METHOD _copyFromModel_SM_ConfigManager
  VAR_IN_OUT
    {attribute 'OPC.UA.DA' := '0'}
    model : M_SM_ConfigManager;
  END_VAR
                  THIS^.proc.save._copyFromModel_WriteXmlProcess( model := model.proc.save );
THIS^.proc.load._copyFromModel_ReadXmlProcess( model := model.proc.load );
THIS^.proc.activate._copyFromModel_ActivateProcess( model := model.proc.activate );

                
END_METHOD

METHOD _copyToModel_SM_ConfigManager
  VAR_IN_OUT
    {attribute 'OPC.UA.DA' := '0'}
    model : M_SM_ConfigManager;
  END_VAR
                  model.filePath := THIS^.filePath;
model.actualStatus := THIS^.actualStatus;
model.stat := THIS^.stat;
THIS^.proc.save._copyToModel_WriteXmlProcess( model := model.proc.save );
THIS^.proc.load._copyToModel_ReadXmlProcess( model := model.proc.load );
THIS^.proc.activate._copyToModel_ActivateProcess( model := model.proc.activate );

                
END_METHOD
END_FUNCTION_BLOCK

FUNCTION_BLOCK SM_ModbusRTUBus
  VAR_INPUT
    {attribute 'OPC.UA.DA' := '1'}
    {attribute 'OPC.UA.DA.Access' := '1'}
    retries : INT := 3;  (* Number of retries for a succesfull process *)
    {attribute 'OPC.UA.DA' := '0'}
    isEnabled : BOOL;  (* Is control enabled? *)
  END_VAR
  VAR_OUTPUT
    {attribute 'OPC.UA.DA' := '1'}
    {attribute 'OPC.UA.DA.Access' := '1'}
    actualStatus : STRING(50);  (* Current status description *)
    {attribute 'OPC.UA.DA' := '1'}
    stat : ModbusRTUBusStatuses;  (* Statuses of the state machine *)
    {attribute 'OPC.UA.DA' := '1'}
    proc : ModbusRTUBusProcesses;  (* Processes of the state machine *)
  END_VAR

            stat.busy := F_BusyStatus(
    superState := TRUE,
    isBusy := proc.readCoil.stat.busy.busy OR (proc.writeCoil.stat.busy.busy OR (proc.readRegister.stat.busy.busy OR (proc.writeRegister.stat.busy.busy OR proc.diagnostics.stat.busy.busy))));
proc.readCoil( isEnabled := isEnabled AND (stat.busy = BusyStatus.idle) );
proc.writeCoil( isEnabled := isEnabled AND (stat.busy = BusyStatus.idle) );
proc.readRegister( isEnabled := isEnabled AND (stat.busy = BusyStatus.idle) );
proc.writeRegister( isEnabled := isEnabled AND (stat.busy = BusyStatus.idle) );
proc.diagnostics( isEnabled := isEnabled AND (stat.busy = BusyStatus.idle) );

          

METHOD _copyFromModel_SM_ModbusRTUBus
  VAR_IN_OUT
    {attribute 'OPC.UA.DA' := '0'}
    model : M_SM_ModbusRTUBus;
  END_VAR
                  THIS^.proc.readCoil._copyFromModel_ModbusRTUBusReadCoilProcess( model := model.proc.readCoil );
THIS^.proc.writeCoil._copyFromModel_ModbusRTUBusWriteCoilProcess( model := model.proc.writeCoil );
THIS^.proc.readRegister._copyFromModel_ModbusRTUBusReadRegisterProcess( model := model.proc.readRegister );
THIS^.proc.writeRegister._copyFromModel_ModbusRTUBusWriteRegisterProcess( model := model.proc.writeRegister );
THIS^.proc.diagnostics._copyFromModel_ModbusRTUBusDiagnosticsProcess( model := model.proc.diagnostics );

                
END_METHOD

METHOD _copyToModel_SM_ModbusRTUBus
  VAR_IN_OUT
    {attribute 'OPC.UA.DA' := '0'}
    model : M_SM_ModbusRTUBus;
  END_VAR
                  model.retries := THIS^.retries;
model.actualStatus := THIS^.actualStatus;
model.stat := THIS^.stat;
THIS^.proc.readCoil._copyToModel_ModbusRTUBusReadCoilProcess( model := model.proc.readCoil );
THIS^.proc.writeCoil._copyToModel_ModbusRTUBusWriteCoilProcess( model := model.proc.writeCoil );
THIS^.proc.readRegister._copyToModel_ModbusRTUBusReadRegisterProcess( model := model.proc.readRegister );
THIS^.proc.writeRegister._copyToModel_ModbusRTUBusWriteRegisterProcess( model := model.proc.writeRegister );
THIS^.proc.diagnostics._copyToModel_ModbusRTUBusDiagnosticsProcess( model := model.proc.diagnostics );

                
END_METHOD
END_FUNCTION_BLOCK

FUNCTION_BLOCK SM_GigECamera
  VAR_INPUT
    {attribute 'OPC.UA.DA' := '1'}
    {attribute 'OPC.UA.DA.Access' := '1'}
    state : ETcVnCameraState;  (* Camera state *)
    {attribute 'OPC.UA.DA' := '1'}
    {attribute 'OPC.UA.DA.Access' := '1'}
    source : GigECameraSources;  (* Camera source *)
  END_VAR
  VAR_OUTPUT
    {attribute 'OPC.UA.DA' := '1'}
    {attribute 'OPC.UA.DA.Access' := '1'}
    actualStatus : STRING(50);  (* Current status description *)
    {attribute 'OPC.UA.DA' := '1'}
    {attribute 'OPC.UA.DA.Access' := '1'}
    frameCounter : UDINT;  (* Number of frames taken *)
    {attribute 'OPC.UA.DA' := '1'}
    {attribute 'OPC.UA.DA.Access' := '1'}
    loopCounter : UDINT;  (* Number of parameter loops done *)
    {attribute 'OPC.UA.DA' := '1'}
    {attribute 'OPC.UA.DA.Access' := '1'}
    loopSuccessCounter : UDINT;  (* Number of successful parameter loops *)
    {attribute 'OPC.UA.DA' := '1'}
    {attribute 'OPC.UA.DA.Access' := '1'}
    channelOpen : BOOL;  (* Is the camera's control channel open? *)
    {attribute 'OPC.UA.DA' := '1'}
    {attribute 'OPC.UA.DA.Access' := '1'}
    acquiring : BOOL;  (* Is the camera acquiring frames? *)
    {attribute 'OPC.UA.DA' := '1'}
    {attribute 'OPC.UA.DA.Access' := '1'}
    actualMultiTriggerNumber : UDINT;  (* Number of triggers sent for the current multi-trigger process *)
    {attribute 'OPC.UA.DA' := '1'}
    {attribute 'OPC.UA.DA.Access' := '1'}
    maxMultiTriggerNumber : UDINT;  (* Maximum number of triggers that will be sent in the current multi-trigger process *)
    {attribute 'OPC.UA.DA' := '1'}
    {attribute 'OPC.UA.DA.Access' := '1'}
    acquisitionFrameRate : LREAL;  (* Acquisition frame rate in Hz *)
    {attribute 'OPC.UA.DA' := '1'}
    {attribute 'OPC.UA.DA.Access' := '1'}
    linkAcquisitionFrameRate : LREAL;  (* Acquisition frame rate in Hz, limited by the link bandwidth *)
    {attribute 'OPC.UA.DA' := '1'}
    {attribute 'OPC.UA.DA.Access' := '1'}
    exposureTime : LREAL;  (* Exposure time in s *)
    {attribute 'OPC.UA.DA' := '1'}
    {attribute 'OPC.UA.DA.Access' := '1'}
    gainSelector : UDINT;  (* Gain selector *)
    {attribute 'OPC.UA.DA' := '1'}
    {attribute 'OPC.UA.DA.Access' := '1'}
    gain : LREAL;  (* Gain (unitless) of the current GainSelector *)
    {attribute 'OPC.UA.DA' := '1'}
    {attribute 'OPC.UA.DA.Access' := '1'}
    gainAnalog : LREAL;  (* Gain (unitless) of the last time GainSelector was set to Analog *)
    {attribute 'OPC.UA.DA' := '1'}
    {attribute 'OPC.UA.DA.Access' := '1'}
    gainDigital : LREAL;  (* Gain (unitless) of the last time GainSelector was set to Digital *)
    {attribute 'OPC.UA.DA' := '1'}
    {attribute 'OPC.UA.DA.Access' := '1'}
    width : UDINT;  (* Width of the frame, in pixels *)
    {attribute 'OPC.UA.DA' := '1'}
    {attribute 'OPC.UA.DA.Access' := '1'}
    height : UDINT;  (* Height of the frame, in pixels *)
    {attribute 'OPC.UA.DA' := '1'}
    {attribute 'OPC.UA.DA.Access' := '1'}
    offsetX : UDINT;  (* Offset of the frame in X direction, in pixels *)
    {attribute 'OPC.UA.DA' := '1'}
    {attribute 'OPC.UA.DA.Access' := '1'}
    offsetY : UDINT;  (* Offset of the frame in Y direction, in pixels *)
    {attribute 'OPC.UA.DA' := '1'}
    {attribute 'OPC.UA.DA.Access' := '1'}
    widthMax : UDINT;  (* Maximum width of the frame, in pixels *)
    {attribute 'OPC.UA.DA' := '1'}
    {attribute 'OPC.UA.DA.Access' := '1'}
    heightMax : UDINT;  (* Maximum height of the frame, in pixels *)
    {attribute 'OPC.UA.DA' := '1'}
    {attribute 'OPC.UA.DA.Access' := '1'}
    binningSelector : UDINT;  (* Binning engine (sensor or FPGA) *)
    {attribute 'OPC.UA.DA' := '1'}
    {attribute 'OPC.UA.DA.Access' := '1'}
    binningHorizontal : UDINT;  (* Horizontal binning *)
    {attribute 'OPC.UA.DA' := '1'}
    {attribute 'OPC.UA.DA.Access' := '1'}
    binningVertical : UDINT;  (* Vertical binning *)
    {attribute 'OPC.UA.DA' := '1'}
    {attribute 'OPC.UA.DA.Access' := '1'}
    triggerMode : UDINT;  (* Trigger mode *)
    {attribute 'OPC.UA.DA' := '1'}
    {attribute 'OPC.UA.DA.Access' := '1'}
    triggerSelector : UDINT;  (* Trigger selector *)
    {attribute 'OPC.UA.DA' := '1'}
    {attribute 'OPC.UA.DA.Access' := '1'}
    acquisitionMode : UDINT;  (* Acquisition mode *)
    {attribute 'OPC.UA.DA' := '1'}
    {attribute 'OPC.UA.DA.Access' := '1'}
    blackLevel : LREAL;  (* Black level (0 .. 511 for 12-bit images) *)
    {attribute 'OPC.UA.DA' := '1'}
    {attribute 'OPC.UA.DA.Access' := '1'}
    blackLevelAuto : UDINT;  (* Black level auto enum *)
    {attribute 'OPC.UA.DA' := '1'}
    {attribute 'OPC.UA.DA.Access' := '1'}
    deviceTemperature : LREAL;  (* Temperature of the camera, in °C *)
    {attribute 'OPC.UA.DA' := '1'}
    stat : GigECameraStatuses;  (* Statuses of the state machine *)
    {attribute 'OPC.UA.DA' := '1'}
    proc : GigECameraProcesses;  (* Processes of the state machine *)
  END_VAR

            stat.health := F_HealthStatus(
    superState := NOT(state = ETcVnCameraState.TCVN_CS_INITIAL),
    isGood := NOT(state = ETcVnCameraState.TCVN_CS_ERROR),
    hasWarning := FALSE);
stat.busy := F_BusyStatus(
    superState := NOT(state = ETcVnCameraState.TCVN_CS_INITIAL),
    isBusy := (state = ETcVnCameraState.TCVN_CS_INITIALIZING) OR ((state = ETcVnCameraState.TCVN_CS_OPENING) OR (state = ETcVnCameraState.TCVN_CS_CLOSING)));
proc.open( isEnabled := (state = ETcVnCameraState.TCVN_CS_INITIAL) OR ((state = ETcVnCameraState.TCVN_CS_INITIALIZED) OR ((state = ETcVnCameraState.TCVN_CS_OPENING) OR (state = ETcVnCameraState.TCVN_CS_OPENED))) );
proc.close( isEnabled := NOT((state = ETcVnCameraState.TCVN_CS_INITIAL) OR (state = ETcVnCameraState.TCVN_CS_INITIALIZED)) );
proc.startAcquiring( isEnabled := ((state = ETcVnCameraState.TCVN_CS_INITIAL) OR ((state = ETcVnCameraState.TCVN_CS_INITIALIZED) OR (state = ETcVnCameraState.TCVN_CS_OPENED))) AND (proc.stopAcquiring.stat.busy = BusyStatus.idle) );
proc.stopAcquiring( isEnabled := NOT((state = ETcVnCameraState.TCVN_CS_INITIAL) OR (state = ETcVnCameraState.TCVN_CS_INITIALIZED)) );
proc.reset( isEnabled := TRUE );
proc.setup( isEnabled := TRUE );
proc.setParam( isEnabled := TRUE );
proc.setParam2( isEnabled := TRUE );
proc.trigger( isEnabled := TRUE );
proc.pulseTrigger( isEnabled := TRUE );
proc.multiTrigger( isEnabled := TRUE );
proc.multiTriggerAbort( isEnabled := proc.multiTrigger.stat.busy = BusyStatus.busy );
proc.setSource( isEnabled := TRUE );

          

METHOD _copyFromModel_SM_GigECamera
  VAR_IN_OUT
    {attribute 'OPC.UA.DA' := '0'}
    model : M_SM_GigECamera;
  END_VAR
                  THIS^.proc.open._copyFromModel_Process( model := model.proc.open );
THIS^.proc.close._copyFromModel_Process( model := model.proc.close );
THIS^.proc.startAcquiring._copyFromModel_Process( model := model.proc.startAcquiring );
THIS^.proc.stopAcquiring._copyFromModel_Process( model := model.proc.stopAcquiring );
THIS^.proc.reset._copyFromModel_Process( model := model.proc.reset );
THIS^.proc.setup._copyFromModel_GigECameraSetupProcess( model := model.proc.setup );
THIS^.proc.setParam._copyFromModel_GigECameraSetParamProcess( model := model.proc.setParam );
THIS^.proc.setParam2._copyFromModel_GigECameraSetParam2Process( model := model.proc.setParam2 );
THIS^.proc.trigger._copyFromModel_Process( model := model.proc.trigger );
THIS^.proc.pulseTrigger._copyFromModel_GigECameraPulseTrigger( model := model.proc.pulseTrigger );
THIS^.proc.multiTrigger._copyFromModel_GigECameraMultiTriggerProcess( model := model.proc.multiTrigger );
THIS^.proc.multiTriggerAbort._copyFromModel_Process( model := model.proc.multiTriggerAbort );
THIS^.proc.setSource._copyFromModel_GigECameraSetSourceProcess( model := model.proc.setSource );

                
END_METHOD

METHOD _copyToModel_SM_GigECamera
  VAR_IN_OUT
    {attribute 'OPC.UA.DA' := '0'}
    model : M_SM_GigECamera;
  END_VAR
                  model.state := THIS^.state;
model.source := THIS^.source;
model.actualStatus := THIS^.actualStatus;
model.frameCounter := THIS^.frameCounter;
model.loopCounter := THIS^.loopCounter;
model.loopSuccessCounter := THIS^.loopSuccessCounter;
model.channelOpen := THIS^.channelOpen;
model.acquiring := THIS^.acquiring;
model.actualMultiTriggerNumber := THIS^.actualMultiTriggerNumber;
model.maxMultiTriggerNumber := THIS^.maxMultiTriggerNumber;
model.acquisitionFrameRate := THIS^.acquisitionFrameRate;
model.linkAcquisitionFrameRate := THIS^.linkAcquisitionFrameRate;
model.exposureTime := THIS^.exposureTime;
model.gainSelector := THIS^.gainSelector;
model.gain := THIS^.gain;
model.gainAnalog := THIS^.gainAnalog;
model.gainDigital := THIS^.gainDigital;
model.width := THIS^.width;
model.height := THIS^.height;
model.offsetX := THIS^.offsetX;
model.offsetY := THIS^.offsetY;
model.widthMax := THIS^.widthMax;
model.heightMax := THIS^.heightMax;
model.binningSelector := THIS^.binningSelector;
model.binningHorizontal := THIS^.binningHorizontal;
model.binningVertical := THIS^.binningVertical;
model.triggerMode := THIS^.triggerMode;
model.triggerSelector := THIS^.triggerSelector;
model.acquisitionMode := THIS^.acquisitionMode;
model.blackLevel := THIS^.blackLevel;
model.blackLevelAuto := THIS^.blackLevelAuto;
model.deviceTemperature := THIS^.deviceTemperature;
model.stat := THIS^.stat;
THIS^.proc.open._copyToModel_Process( model := model.proc.open );
THIS^.proc.close._copyToModel_Process( model := model.proc.close );
THIS^.proc.startAcquiring._copyToModel_Process( model := model.proc.startAcquiring );
THIS^.proc.stopAcquiring._copyToModel_Process( model := model.proc.stopAcquiring );
THIS^.proc.reset._copyToModel_Process( model := model.proc.reset );
THIS^.proc.setup._copyToModel_GigECameraSetupProcess( model := model.proc.setup );
THIS^.proc.setParam._copyToModel_GigECameraSetParamProcess( model := model.proc.setParam );
THIS^.proc.setParam2._copyToModel_GigECameraSetParam2Process( model := model.proc.setParam2 );
THIS^.proc.trigger._copyToModel_Process( model := model.proc.trigger );
THIS^.proc.pulseTrigger._copyToModel_GigECameraPulseTrigger( model := model.proc.pulseTrigger );
THIS^.proc.multiTrigger._copyToModel_GigECameraMultiTriggerProcess( model := model.proc.multiTrigger );
THIS^.proc.multiTriggerAbort._copyToModel_Process( model := model.proc.multiTriggerAbort );
THIS^.proc.setSource._copyToModel_GigECameraSetSourceProcess( model := model.proc.setSource );

                
END_METHOD
END_FUNCTION_BLOCK

FUNCTION_BLOCK SM_ELL14Stage
  VAR_INPUT
    {attribute 'OPC.UA.DA' := '1'}
    {attribute 'OPC.UA.DA.Access' := '1'}
    simulated : BOOL;  (* True if the device must be simulated *)
    {attribute 'OPC.UA.DA' := '0'}
    isEnabled : BOOL;  (* Is control enabled? *)
  END_VAR
  VAR_OUTPUT
    {attribute 'OPC.UA.DA' := '1'}
    {attribute 'OPC.UA.DA.Access' := '1'}
    actualStatus : STRING(50);  (* Current status description *)
    {attribute 'OPC.UA.DA' := '1'}
    {attribute 'OPC.UA.DA.Access' := '1'}
    commError : BOOL;  (* True if the communication is in error *)
    {attribute 'OPC.UA.DA' := '1'}
    {attribute 'OPC.UA.DA.Access' := '1'}
    homed : BOOL;  (* True if the stage was homed *)
    {attribute 'OPC.UA.DA' := '1'}
    {attribute 'OPC.UA.DA.Access' := '1'}
    position : LREAL;  (* Actual position in ° *)
    {attribute 'OPC.UA.DA' := '1'}
    {attribute 'OPC.UA.DA.Access' := '1'}
    statusCode : ELL14StatusCode;  (* Actual status *)
    {attribute 'OPC.UA.DA' := '1'}
    stat : ELL14StageStatuses;  (* Statuses of the state machine *)
    {attribute 'OPC.UA.DA' := '1'}
    proc : ELL14StageProcesses;  (* Processes of the state machine *)
  END_VAR

            stat.health := F_HealthStatus(
    superState := TRUE,
    hasWarning := FALSE,
    isGood := (NOT(commError)) AND ((statusCode = ELL14StatusCode.OK) OR (statusCode = ELL14StatusCode.BUSY)));
stat.busy := F_BusyStatus(
    superState := TRUE,
    isBusy := statusCode = ELL14StatusCode.BUSY);
proc.moveAbs( isEnabled := isEnabled AND homed );
proc.moveRel( isEnabled := isEnabled AND homed );
proc.send( isEnabled := isEnabled );

          

METHOD _copyFromModel_SM_ELL14Stage
  VAR_IN_OUT
    {attribute 'OPC.UA.DA' := '0'}
    model : M_SM_ELL14Stage;
  END_VAR
                  THIS^.proc.moveAbs._copyFromModel_Arg1LrealProcess( model := model.proc.moveAbs );
THIS^.proc.moveRel._copyFromModel_Arg1LrealProcess( model := model.proc.moveRel );
THIS^.proc.send._copyFromModel_Ell114SendProcess( model := model.proc.send );

                
END_METHOD

METHOD _copyToModel_SM_ELL14Stage
  VAR_IN_OUT
    {attribute 'OPC.UA.DA' := '0'}
    model : M_SM_ELL14Stage;
  END_VAR
                  model.simulated := THIS^.simulated;
model.actualStatus := THIS^.actualStatus;
model.commError := THIS^.commError;
model.homed := THIS^.homed;
model.position := THIS^.position;
model.statusCode := THIS^.statusCode;
model.stat := THIS^.stat;
THIS^.proc.moveAbs._copyToModel_Arg1LrealProcess( model := model.proc.moveAbs );
THIS^.proc.moveRel._copyToModel_Arg1LrealProcess( model := model.proc.moveRel );
THIS^.proc.send._copyToModel_Ell114SendProcess( model := model.proc.send );

                
END_METHOD
END_FUNCTION_BLOCK

FUNCTION_BLOCK SM_Sequencer
  VAR_INPUT
    {attribute 'OPC.UA.DA' := '1'}
    {attribute 'OPC.UA.DA.Access' := '3'}
    editableSeq : SequenceEnumConfig_M;  (* Editable sequence *)
    {attribute 'OPC.UA.DA' := '0'}
    isEnabled : BOOL;  (* Is control enabled? *)
  END_VAR
  VAR_OUTPUT
    {attribute 'OPC.UA.DA' := '1'}
    {attribute 'OPC.UA.DA.Access' := '1'}
    actualStatus : STRING(50);  (* Current status description *)
    {attribute 'OPC.UA.DA' := '1'}
    {attribute 'OPC.UA.DA.Access' := '1'}
    runnableSeq : SequenceEnumConfig_M;  (* Currently selected sequence for running *)
    {attribute 'OPC.UA.DA' := '1'}
    {attribute 'OPC.UA.DA.Access' := '1'}
    runnableStat : ARRAY[0..29] OF ActionStatus;  (* Statuses of the currently selected sequence for running *)
    {attribute 'OPC.UA.DA' := '1'}
    {attribute 'OPC.UA.DA.Access' := '1'}
    runnableIndex : UINT;  (* Index of the currently selected sequence for running *)
    {attribute 'OPC.UA.DA' := '1'}
    {attribute 'OPC.UA.DA.Access' := '1'}
    editableIndex : UINT;  (* Index of the currently selected sequence for editing *)
    {attribute 'OPC.UA.DA' := '1'}
    {attribute 'OPC.UA.DA.Access' := '1'}
    ids : ARRAY[0..50] OF STRING(30);  (* Available IDs *)
    {attribute 'OPC.UA.DA' := '1'}
    stat : SequencerStatuses;  (* Statuses of the state machine *)
    {attribute 'OPC.UA.DA' := '1'}
    parts : SequencerParts;  (* Parts of the state machine *)
    {attribute 'OPC.UA.DA' := '1'}
    proc : SequencerProcesses;  (* Processes of the state machine *)
  END_VAR
  VAR
    {attribute 'OPC.UA.DA' := '0'}
    isError : BOOL;  (* Error present *)
    {attribute 'OPC.UA.DA' := '0'}
    isBusy : BOOL;  (* Error present *)
    {attribute 'OPC.UA.DA' := '0'}
    activeConfig : SequencerStringConfig;  (* Active config to be serialized to/from *)
    {attribute 'OPC.UA.DA' := '0'}
    editableConfig : SequencerStringConfig;  (* Editable config to be serialized to/from *)
  END_VAR

            parts.configManager( isEnabled := isEnabled AND (stat.busy = BusyStatus.idle) );
stat.health := F_HealthStatus(
    superState := TRUE,
    hasWarning := FALSE,
    isGood := NOT(isError));
stat.busy := F_BusyStatus(
    superState := TRUE,
    isBusy := isBusy OR (parts.configManager.stat.busy = BusyStatus.busy));
proc.selectEditable( isEnabled := isEnabled AND (stat.busy = BusyStatus.idle) );
proc.selectRunnable( isEnabled := isEnabled AND (stat.busy = BusyStatus.idle) );
proc.start( isEnabled := isEnabled AND (stat.busy = BusyStatus.idle) );
proc.stop( isEnabled := isEnabled AND (stat.busy = BusyStatus.busy) );
proc.apply( isEnabled := isEnabled AND (stat.busy = BusyStatus.idle) );
proc.cancel();

          

METHOD _copyFromModel_SM_Sequencer
  VAR_IN_OUT
    {attribute 'OPC.UA.DA' := '0'}
    model : M_SM_Sequencer;
  END_VAR
                  THIS^.editableSeq := model.editableSeq;
THIS^.parts.configManager._copyFromModel_ConfigManager( model := model.parts.configManager );
THIS^.proc.selectEditable._copyFromModel_IndexProcess( model := model.proc.selectEditable );
THIS^.proc.selectRunnable._copyFromModel_IndexProcess( model := model.proc.selectRunnable );
THIS^.proc.start._copyFromModel_IdProcess( model := model.proc.start );
THIS^.proc.stop._copyFromModel_Process( model := model.proc.stop );
THIS^.proc.apply._copyFromModel_Process( model := model.proc.apply );
THIS^.proc.cancel._copyFromModel_Process( model := model.proc.cancel );

                
END_METHOD

METHOD _copyToModel_SM_Sequencer
  VAR_IN_OUT
    {attribute 'OPC.UA.DA' := '0'}
    model : M_SM_Sequencer;
  END_VAR
                  model.editableSeq := THIS^.editableSeq;
model.actualStatus := THIS^.actualStatus;
model.runnableSeq := THIS^.runnableSeq;
model.runnableStat := THIS^.runnableStat;
model.runnableIndex := THIS^.runnableIndex;
model.editableIndex := THIS^.editableIndex;
model.ids := THIS^.ids;
model.stat := THIS^.stat;
THIS^.parts.configManager._copyToModel_ConfigManager( model := model.parts.configManager );
THIS^.proc.selectEditable._copyToModel_IndexProcess( model := model.proc.selectEditable );
THIS^.proc.selectRunnable._copyToModel_IndexProcess( model := model.proc.selectRunnable );
THIS^.proc.start._copyToModel_IdProcess( model := model.proc.start );
THIS^.proc.stop._copyToModel_Process( model := model.proc.stop );
THIS^.proc.apply._copyToModel_Process( model := model.proc.apply );
THIS^.proc.cancel._copyToModel_Process( model := model.proc.cancel );

                
END_METHOD
END_FUNCTION_BLOCK

FUNCTION_BLOCK SM_EventManager
  VAR_OUTPUT
    {attribute 'OPC.UA.DA' := '1'}
    {attribute 'OPC.UA.DA.Access' := '1'}
    actualStatus : STRING(50);  (* Current status description *)
    {attribute 'OPC.UA.DA' := '1'}
    {attribute 'OPC.UA.DA.Access' := '1'}
    alarmCount : INT;  (* Number of alarms *)
    {attribute 'OPC.UA.DA' := '1'}
    stat : EventManagerStatuses;  (* Statuses of the state machine *)
  END_VAR

            
          

METHOD _copyFromModel_SM_EventManager
  VAR_IN_OUT
    {attribute 'OPC.UA.DA' := '0'}
    model : M_SM_EventManager;
  END_VAR
                  
                
END_METHOD

METHOD _copyToModel_SM_EventManager
  VAR_IN_OUT
    {attribute 'OPC.UA.DA' := '0'}
    model : M_SM_EventManager;
  END_VAR
                  model.actualStatus := THIS^.actualStatus;
model.alarmCount := THIS^.alarmCount;
model.stat := THIS^.stat;

                
END_METHOD
END_FUNCTION_BLOCK

FUNCTION_BLOCK Process EXTENDS BaseProcess

            IF do_request OR atomic.request THEN
    do_request_result := request();
    do_request := FALSE;
    atomic.request := FALSE;
END_IF;
SUPER^();

          

{attribute 'TcRpcEnable' := '1'}
METHOD start
                  IF THIS^.atomic.request THEN
    THIS^.stat.handle := THIS^.atomic.handle;
ELSE
    THIS^.stat.handle := 0;
END_IF;
THIS^.stat.busy := BusyStatus.busy;
THIS^.stat.health := HealthStatus.good;

                
END_METHOD

{attribute 'TcRpcEnable' := '1'}
METHOD request : RequestResults
                  IF THIS^.stat.enabled = EnabledStatus.enabled THEN
    request := RequestResults.ACCEPTED;
    THIS^.start();
ELSE
    request := RequestResults.REJECTED;
    IF THIS^.atomic.request THEN
        THIS^.lastRejectedHandle := THIS^.atomic.handle;
    END_IF;
END_IF;

                
END_METHOD

METHOD _copyFromModel_Process
  VAR_IN_OUT
    {attribute 'OPC.UA.DA' := '0'}
    model : M_Process;
  END_VAR
                  SUPER^._copyFromModel_BaseProcess( model := model );

                
END_METHOD

METHOD _copyToModel_Process
  VAR_IN_OUT
    {attribute 'OPC.UA.DA' := '0'}
    model : M_Process;
  END_VAR
                  SUPER^._copyToModel_BaseProcess( model := model );

                
END_METHOD
END_FUNCTION_BLOCK

FUNCTION_BLOCK IdProcess EXTENDS BaseProcess
  VAR_INPUT
    {attribute 'OPC.UA.DA' := '1'}
    {attribute 'OPC.UA.DA.Access' := '3'}
    {attribute 'TcHmiSymbol.Show'}
    set : IdProcessArgs;  (* Arguments to be set, before writing do_request TRUE *)
  END_VAR
  VAR_OUTPUT
    {attribute 'OPC.UA.DA' := '0'}
    get : IdProcessArgs;  (* Arguments in use by the process, if do_request was accepted *)
  END_VAR

            IF do_request OR atomic.request THEN
    do_request_result := request( id := set.id );
    do_request := FALSE;
    atomic.request := FALSE;
END_IF;
SUPER^();

          

{attribute 'TcRpcEnable' := '1'}
METHOD start
  VAR_INPUT
    id : STRING(30);
  END_VAR
                  THIS^.get.id := id;
IF THIS^.atomic.request THEN
    THIS^.stat.handle := THIS^.atomic.handle;
ELSE
    THIS^.stat.handle := 0;
END_IF;
THIS^.stat.busy := BusyStatus.busy;
THIS^.stat.health := HealthStatus.good;

                
END_METHOD

{attribute 'TcRpcEnable' := '1'}
METHOD request : RequestResults
  VAR_INPUT
    id : STRING(30);
  END_VAR
                  IF THIS^.stat.enabled = EnabledStatus.enabled THEN
    request := RequestResults.ACCEPTED;
    THIS^.start( id := id );
ELSE
    request := RequestResults.REJECTED;
    IF THIS^.atomic.request THEN
        THIS^.lastRejectedHandle := THIS^.atomic.handle;
    END_IF;
END_IF;

                
END_METHOD

METHOD _copyFromModel_IdProcess
  VAR_IN_OUT
    {attribute 'OPC.UA.DA' := '0'}
    model : M_IdProcess;
  END_VAR
                  THIS^.set := model.set;
SUPER^._copyFromModel_BaseProcess( model := model );

                
END_METHOD

METHOD _copyToModel_IdProcess
  VAR_IN_OUT
    {attribute 'OPC.UA.DA' := '0'}
    model : M_IdProcess;
  END_VAR
                  model.set := THIS^.set;
SUPER^._copyToModel_BaseProcess( model := model );

                
END_METHOD
END_FUNCTION_BLOCK

FUNCTION_BLOCK IndexProcess EXTENDS BaseProcess
  VAR_INPUT
    {attribute 'OPC.UA.DA' := '1'}
    {attribute 'OPC.UA.DA.Access' := '3'}
    {attribute 'TcHmiSymbol.Show'}
    set : IndexProcessArgs;  (* Arguments to be set, before writing do_request TRUE *)
  END_VAR
  VAR_OUTPUT
    {attribute 'OPC.UA.DA' := '0'}
    get : IndexProcessArgs;  (* Arguments in use by the process, if do_request was accepted *)
  END_VAR

            IF do_request OR atomic.request THEN
    do_request_result := request( id := set.id );
    do_request := FALSE;
    atomic.request := FALSE;
END_IF;
SUPER^();

          

{attribute 'TcRpcEnable' := '1'}
METHOD start
  VAR_INPUT
    id : UINT;
  END_VAR
                  THIS^.get.id := id;
IF THIS^.atomic.request THEN
    THIS^.stat.handle := THIS^.atomic.handle;
ELSE
    THIS^.stat.handle := 0;
END_IF;
THIS^.stat.busy := BusyStatus.busy;
THIS^.stat.health := HealthStatus.good;

                
END_METHOD

{attribute 'TcRpcEnable' := '1'}
METHOD request : RequestResults
  VAR_INPUT
    id : UINT;
  END_VAR
                  IF THIS^.stat.enabled = EnabledStatus.enabled THEN
    request := RequestResults.ACCEPTED;
    THIS^.start( id := id );
ELSE
    request := RequestResults.REJECTED;
    IF THIS^.atomic.request THEN
        THIS^.lastRejectedHandle := THIS^.atomic.handle;
    END_IF;
END_IF;

                
END_METHOD

METHOD _copyFromModel_IndexProcess
  VAR_IN_OUT
    {attribute 'OPC.UA.DA' := '0'}
    model : M_IndexProcess;
  END_VAR
                  THIS^.set := model.set;
SUPER^._copyFromModel_BaseProcess( model := model );

                
END_METHOD

METHOD _copyToModel_IndexProcess
  VAR_IN_OUT
    {attribute 'OPC.UA.DA' := '0'}
    model : M_IndexProcess;
  END_VAR
                  model.set := THIS^.set;
SUPER^._copyToModel_BaseProcess( model := model );

                
END_METHOD
END_FUNCTION_BLOCK

FUNCTION_BLOCK McProcess EXTENDS BaseMcProcess

            IF do_request OR atomic.request THEN
    do_request_result := request();
    do_request := FALSE;
    atomic.request := FALSE;
END_IF;
SUPER^();

          

{attribute 'TcRpcEnable' := '1'}
METHOD start
                  IF THIS^.atomic.request THEN
    THIS^.stat.handle := THIS^.atomic.handle;
ELSE
    THIS^.stat.handle := 0;
END_IF;
THIS^.stat.busy := BusyStatus.busy;
THIS^.stat.health := HealthStatus.good;

                
END_METHOD

{attribute 'TcRpcEnable' := '1'}
METHOD request : RequestResults
                  IF THIS^.stat.enabled = EnabledStatus.enabled THEN
    request := RequestResults.ACCEPTED;
    THIS^.start();
ELSE
    request := RequestResults.REJECTED;
    IF THIS^.atomic.request THEN
        THIS^.lastRejectedHandle := THIS^.atomic.handle;
    END_IF;
END_IF;

                
END_METHOD

METHOD _copyFromModel_McProcess
  VAR_IN_OUT
    {attribute 'OPC.UA.DA' := '0'}
    model : M_McProcess;
  END_VAR
                  SUPER^._copyFromModel_BaseMcProcess( model := model );

                
END_METHOD

METHOD _copyToModel_McProcess
  VAR_IN_OUT
    {attribute 'OPC.UA.DA' := '0'}
    model : M_McProcess;
  END_VAR
                  SUPER^._copyToModel_BaseMcProcess( model := model );

                
END_METHOD
END_FUNCTION_BLOCK

FUNCTION_BLOCK ChangeSetpointProcess EXTENDS BaseProcess
  VAR_INPUT
    {attribute 'OPC.UA.DA' := '1'}
    {attribute 'OPC.UA.DA.Access' := '3'}
    {attribute 'TcHmiSymbol.Show'}
    set : ChangeSetpointProcessArgs;  (* Arguments to be set, before writing do_request TRUE *)
  END_VAR
  VAR_OUTPUT
    {attribute 'OPC.UA.DA' := '0'}
    get : ChangeSetpointProcessArgs;  (* Arguments in use by the process, if do_request was accepted *)
  END_VAR

            IF do_request OR atomic.request THEN
    do_request_result := request( setpoint := set.setpoint );
    do_request := FALSE;
    atomic.request := FALSE;
END_IF;
SUPER^();

          

{attribute 'TcRpcEnable' := '1'}
METHOD start
  VAR_INPUT
    setpoint : LREAL;  (* New setpoint value *)
  END_VAR
                  THIS^.get.setpoint := setpoint;
IF THIS^.atomic.request THEN
    THIS^.stat.handle := THIS^.atomic.handle;
ELSE
    THIS^.stat.handle := 0;
END_IF;
THIS^.stat.busy := BusyStatus.busy;
THIS^.stat.health := HealthStatus.good;

                
END_METHOD

{attribute 'TcRpcEnable' := '1'}
METHOD request : RequestResults
  VAR_INPUT
    setpoint : LREAL;  (* New setpoint value *)
  END_VAR
                  IF THIS^.stat.enabled = EnabledStatus.enabled THEN
    request := RequestResults.ACCEPTED;
    THIS^.start( setpoint := setpoint );
ELSE
    request := RequestResults.REJECTED;
    IF THIS^.atomic.request THEN
        THIS^.lastRejectedHandle := THIS^.atomic.handle;
    END_IF;
END_IF;

                
END_METHOD

METHOD _copyFromModel_ChangeSetpointProcess
  VAR_IN_OUT
    {attribute 'OPC.UA.DA' := '0'}
    model : M_ChangeSetpointProcess;
  END_VAR
                  THIS^.set := model.set;
SUPER^._copyFromModel_BaseProcess( model := model );

                
END_METHOD

METHOD _copyToModel_ChangeSetpointProcess
  VAR_IN_OUT
    {attribute 'OPC.UA.DA' := '0'}
    model : M_ChangeSetpointProcess;
  END_VAR
                  model.set := THIS^.set;
SUPER^._copyToModel_BaseProcess( model := model );

                
END_METHOD
END_FUNCTION_BLOCK

FUNCTION_BLOCK ChangeParameterProcess EXTENDS BaseProcess
  VAR_INPUT
    {attribute 'OPC.UA.DA' := '1'}
    {attribute 'OPC.UA.DA.Access' := '3'}
    {attribute 'TcHmiSymbol.Show'}
    set : ChangeParameterProcessArgs;  (* Arguments to be set, before writing do_request TRUE *)
  END_VAR
  VAR_OUTPUT
    {attribute 'OPC.UA.DA' := '0'}
    get : ChangeParameterProcessArgs;  (* Arguments in use by the process, if do_request was accepted *)
  END_VAR

            IF do_request OR atomic.request THEN
    do_request_result := request( parameter := set.parameter );
    do_request := FALSE;
    atomic.request := FALSE;
END_IF;
SUPER^();

          

{attribute 'TcRpcEnable' := '1'}
METHOD start
  VAR_INPUT
    parameter : LREAL;  (* New parameter value *)
  END_VAR
                  THIS^.get.parameter := parameter;
IF THIS^.atomic.request THEN
    THIS^.stat.handle := THIS^.atomic.handle;
ELSE
    THIS^.stat.handle := 0;
END_IF;
THIS^.stat.busy := BusyStatus.busy;
THIS^.stat.health := HealthStatus.good;

                
END_METHOD

{attribute 'TcRpcEnable' := '1'}
METHOD request : RequestResults
  VAR_INPUT
    parameter : LREAL;  (* New parameter value *)
  END_VAR
                  IF THIS^.stat.enabled = EnabledStatus.enabled THEN
    request := RequestResults.ACCEPTED;
    THIS^.start( parameter := parameter );
ELSE
    request := RequestResults.REJECTED;
    IF THIS^.atomic.request THEN
        THIS^.lastRejectedHandle := THIS^.atomic.handle;
    END_IF;
END_IF;

                
END_METHOD

METHOD _copyFromModel_ChangeParameterProcess
  VAR_IN_OUT
    {attribute 'OPC.UA.DA' := '0'}
    model : M_ChangeParameterProcess;
  END_VAR
                  THIS^.set := model.set;
SUPER^._copyFromModel_BaseProcess( model := model );

                
END_METHOD

METHOD _copyToModel_ChangeParameterProcess
  VAR_IN_OUT
    {attribute 'OPC.UA.DA' := '0'}
    model : M_ChangeParameterProcess;
  END_VAR
                  model.set := THIS^.set;
SUPER^._copyToModel_BaseProcess( model := model );

                
END_METHOD
END_FUNCTION_BLOCK

FUNCTION_BLOCK McMoveAbsoluteProcess EXTENDS BaseMcProcess
  VAR_INPUT
    {attribute 'OPC.UA.DA' := '1'}
    {attribute 'OPC.UA.DA.Access' := '3'}
    {attribute 'TcHmiSymbol.Show'}
    set : McMoveAbsoluteProcessArgs;  (* Arguments to be set, before writing do_request TRUE *)
  END_VAR
  VAR_OUTPUT
    {attribute 'OPC.UA.DA' := '0'}
    get : McMoveAbsoluteProcessArgs;  (* Arguments in use by the process, if do_request was accepted *)
  END_VAR

            IF do_request OR atomic.request THEN
    do_request_result := request(
    position := set.position,
    maxVelocity := set.maxVelocity);
    do_request := FALSE;
    atomic.request := FALSE;
END_IF;
SUPER^();

          

{attribute 'TcRpcEnable' := '1'}
METHOD start
  VAR_INPUT
    position : LREAL;  (* New position setpoint *)
    maxVelocity : LREAL;  (* Maximum velocity *)
  END_VAR
                  THIS^.get.position := position;
THIS^.get.maxVelocity := maxVelocity;
IF THIS^.atomic.request THEN
    THIS^.stat.handle := THIS^.atomic.handle;
ELSE
    THIS^.stat.handle := 0;
END_IF;
THIS^.stat.busy := BusyStatus.busy;
THIS^.stat.health := HealthStatus.good;

                
END_METHOD

{attribute 'TcRpcEnable' := '1'}
METHOD request : RequestResults
  VAR_INPUT
    position : LREAL;  (* New position setpoint *)
    maxVelocity : LREAL;  (* Maximum velocity *)
  END_VAR
                  IF THIS^.stat.enabled = EnabledStatus.enabled THEN
    request := RequestResults.ACCEPTED;
    THIS^.start(
        position := position,
        maxVelocity := maxVelocity);
ELSE
    request := RequestResults.REJECTED;
    IF THIS^.atomic.request THEN
        THIS^.lastRejectedHandle := THIS^.atomic.handle;
    END_IF;
END_IF;

                
END_METHOD

METHOD _copyFromModel_McMoveAbsoluteProcess
  VAR_IN_OUT
    {attribute 'OPC.UA.DA' := '0'}
    model : M_McMoveAbsoluteProcess;
  END_VAR
                  THIS^.set := model.set;
SUPER^._copyFromModel_BaseMcProcess( model := model );

                
END_METHOD

METHOD _copyToModel_McMoveAbsoluteProcess
  VAR_IN_OUT
    {attribute 'OPC.UA.DA' := '0'}
    model : M_McMoveAbsoluteProcess;
  END_VAR
                  model.set := THIS^.set;
SUPER^._copyToModel_BaseMcProcess( model := model );

                
END_METHOD
END_FUNCTION_BLOCK

FUNCTION_BLOCK McMoveRelativeProcess EXTENDS BaseMcProcess
  VAR_INPUT
    {attribute 'OPC.UA.DA' := '1'}
    {attribute 'OPC.UA.DA.Access' := '3'}
    {attribute 'TcHmiSymbol.Show'}
    set : McMoveRelativeProcessArgs;  (* Arguments to be set, before writing do_request TRUE *)
  END_VAR
  VAR_OUTPUT
    {attribute 'OPC.UA.DA' := '0'}
    get : McMoveRelativeProcessArgs;  (* Arguments in use by the process, if do_request was accepted *)
  END_VAR

            IF do_request OR atomic.request THEN
    do_request_result := request(
    distance := set.distance,
    maxVelocity := set.maxVelocity);
    do_request := FALSE;
    atomic.request := FALSE;
END_IF;
SUPER^();

          

{attribute 'TcRpcEnable' := '1'}
METHOD start
  VAR_INPUT
    distance : LREAL;  (* Distance to move *)
    maxVelocity : LREAL;  (* Maximum velocity *)
  END_VAR
                  THIS^.get.distance := distance;
THIS^.get.maxVelocity := maxVelocity;
IF THIS^.atomic.request THEN
    THIS^.stat.handle := THIS^.atomic.handle;
ELSE
    THIS^.stat.handle := 0;
END_IF;
THIS^.stat.busy := BusyStatus.busy;
THIS^.stat.health := HealthStatus.good;

                
END_METHOD

{attribute 'TcRpcEnable' := '1'}
METHOD request : RequestResults
  VAR_INPUT
    distance : LREAL;  (* Distance to move *)
    maxVelocity : LREAL;  (* Maximum velocity *)
  END_VAR
                  IF THIS^.stat.enabled = EnabledStatus.enabled THEN
    request := RequestResults.ACCEPTED;
    THIS^.start(
        distance := distance,
        maxVelocity := maxVelocity);
ELSE
    request := RequestResults.REJECTED;
    IF THIS^.atomic.request THEN
        THIS^.lastRejectedHandle := THIS^.atomic.handle;
    END_IF;
END_IF;

                
END_METHOD

METHOD _copyFromModel_McMoveRelativeProcess
  VAR_IN_OUT
    {attribute 'OPC.UA.DA' := '0'}
    model : M_McMoveRelativeProcess;
  END_VAR
                  THIS^.set := model.set;
SUPER^._copyFromModel_BaseMcProcess( model := model );

                
END_METHOD

METHOD _copyToModel_McMoveRelativeProcess
  VAR_IN_OUT
    {attribute 'OPC.UA.DA' := '0'}
    model : M_McMoveRelativeProcess;
  END_VAR
                  model.set := THIS^.set;
SUPER^._copyToModel_BaseMcProcess( model := model );

                
END_METHOD
END_FUNCTION_BLOCK

FUNCTION_BLOCK McPowerProcess EXTENDS BaseMcProcess
  VAR_INPUT
    {attribute 'OPC.UA.DA' := '1'}
    {attribute 'OPC.UA.DA.Access' := '3'}
    {attribute 'TcHmiSymbol.Show'}
    set : McPowerProcessArgs;  (* Arguments to be set, before writing do_request TRUE *)
  END_VAR
  VAR_OUTPUT
    {attribute 'OPC.UA.DA' := '0'}
    get : McPowerProcessArgs;  (* Arguments in use by the process, if do_request was accepted *)
  END_VAR

            IF do_request OR atomic.request THEN
    do_request_result := request( enable := set.enable );
    do_request := FALSE;
    atomic.request := FALSE;
END_IF;
SUPER^();

          

{attribute 'TcRpcEnable' := '1'}
METHOD start
  VAR_INPUT
    enable : BOOL;  (* Enable the power or not *)
  END_VAR
                  THIS^.get.enable := enable;
IF THIS^.atomic.request THEN
    THIS^.stat.handle := THIS^.atomic.handle;
ELSE
    THIS^.stat.handle := 0;
END_IF;
THIS^.stat.busy := BusyStatus.busy;
THIS^.stat.health := HealthStatus.good;

                
END_METHOD

{attribute 'TcRpcEnable' := '1'}
METHOD request : RequestResults
  VAR_INPUT
    enable : BOOL;  (* Enable the power or not *)
  END_VAR
                  IF THIS^.stat.enabled = EnabledStatus.enabled THEN
    request := RequestResults.ACCEPTED;
    THIS^.start( enable := enable );
ELSE
    request := RequestResults.REJECTED;
    IF THIS^.atomic.request THEN
        THIS^.lastRejectedHandle := THIS^.atomic.handle;
    END_IF;
END_IF;

                
END_METHOD

METHOD _copyFromModel_McPowerProcess
  VAR_IN_OUT
    {attribute 'OPC.UA.DA' := '0'}
    model : M_McPowerProcess;
  END_VAR
                  THIS^.set := model.set;
SUPER^._copyFromModel_BaseMcProcess( model := model );

                
END_METHOD

METHOD _copyToModel_McPowerProcess
  VAR_IN_OUT
    {attribute 'OPC.UA.DA' := '0'}
    model : M_McPowerProcess;
  END_VAR
                  model.set := THIS^.set;
SUPER^._copyToModel_BaseMcProcess( model := model );

                
END_METHOD
END_FUNCTION_BLOCK

FUNCTION_BLOCK McSetPositionProcess EXTENDS BaseMcProcess
  VAR_INPUT
    {attribute 'OPC.UA.DA' := '1'}
    {attribute 'OPC.UA.DA.Access' := '3'}
    {attribute 'TcHmiSymbol.Show'}
    set : McSetPositionProcessArgs;  (* Arguments to be set, before writing do_request TRUE *)
  END_VAR
  VAR_OUTPUT
    {attribute 'OPC.UA.DA' := '0'}
    get : McSetPositionProcessArgs;  (* Arguments in use by the process, if do_request was accepted *)
  END_VAR

            IF do_request OR atomic.request THEN
    do_request_result := request( value := set.value );
    do_request := FALSE;
    atomic.request := FALSE;
END_IF;
SUPER^();

          

{attribute 'TcRpcEnable' := '1'}
METHOD start
  VAR_INPUT
    value : LREAL;  (* New position to be taken over by the encoder *)
  END_VAR
                  THIS^.get.value := value;
IF THIS^.atomic.request THEN
    THIS^.stat.handle := THIS^.atomic.handle;
ELSE
    THIS^.stat.handle := 0;
END_IF;
THIS^.stat.busy := BusyStatus.busy;
THIS^.stat.health := HealthStatus.good;

                
END_METHOD

{attribute 'TcRpcEnable' := '1'}
METHOD request : RequestResults
  VAR_INPUT
    value : LREAL;  (* New position to be taken over by the encoder *)
  END_VAR
                  IF THIS^.stat.enabled = EnabledStatus.enabled THEN
    request := RequestResults.ACCEPTED;
    THIS^.start( value := value );
ELSE
    request := RequestResults.REJECTED;
    IF THIS^.atomic.request THEN
        THIS^.lastRejectedHandle := THIS^.atomic.handle;
    END_IF;
END_IF;

                
END_METHOD

METHOD _copyFromModel_McSetPositionProcess
  VAR_IN_OUT
    {attribute 'OPC.UA.DA' := '0'}
    model : M_McSetPositionProcess;
  END_VAR
                  THIS^.set := model.set;
SUPER^._copyFromModel_BaseMcProcess( model := model );

                
END_METHOD

METHOD _copyToModel_McSetPositionProcess
  VAR_IN_OUT
    {attribute 'OPC.UA.DA' := '0'}
    model : M_McSetPositionProcess;
  END_VAR
                  model.set := THIS^.set;
SUPER^._copyToModel_BaseMcProcess( model := model );

                
END_METHOD
END_FUNCTION_BLOCK

FUNCTION_BLOCK McStopProcess EXTENDS BaseMcProcess
  VAR_INPUT
    {attribute 'OPC.UA.DA' := '1'}
    {attribute 'OPC.UA.DA.Access' := '3'}
    {attribute 'TcHmiSymbol.Show'}
    set : McStopProcessArgs;  (* Arguments to be set, before writing do_request TRUE *)
  END_VAR
  VAR_OUTPUT
    {attribute 'OPC.UA.DA' := '0'}
    get : McStopProcessArgs;  (* Arguments in use by the process, if do_request was accepted *)
  END_VAR

            IF do_request OR atomic.request THEN
    do_request_result := request(
    deceleration := set.deceleration,
    jerk := set.jerk);
    do_request := FALSE;
    atomic.request := FALSE;
END_IF;
SUPER^();

          

{attribute 'TcRpcEnable' := '1'}
METHOD start
  VAR_INPUT
    deceleration : LREAL;  (* Deceleration (use 0 for default). If non zero, then also jerk must be non zero! *)
    jerk : LREAL;  (* Jerk (use 0 for default). If non zero, then also deceleration must be non zero! *)
  END_VAR
                  THIS^.get.deceleration := deceleration;
THIS^.get.jerk := jerk;
IF THIS^.atomic.request THEN
    THIS^.stat.handle := THIS^.atomic.handle;
ELSE
    THIS^.stat.handle := 0;
END_IF;
THIS^.stat.busy := BusyStatus.busy;
THIS^.stat.health := HealthStatus.good;

                
END_METHOD

{attribute 'TcRpcEnable' := '1'}
METHOD request : RequestResults
  VAR_INPUT
    deceleration : LREAL;  (* Deceleration (use 0 for default). If non zero, then also jerk must be non zero! *)
    jerk : LREAL;  (* Jerk (use 0 for default). If non zero, then also deceleration must be non zero! *)
  END_VAR
                  IF THIS^.stat.enabled = EnabledStatus.enabled THEN
    request := RequestResults.ACCEPTED;
    THIS^.start(
        deceleration := deceleration,
        jerk := jerk);
ELSE
    request := RequestResults.REJECTED;
    IF THIS^.atomic.request THEN
        THIS^.lastRejectedHandle := THIS^.atomic.handle;
    END_IF;
END_IF;

                
END_METHOD

METHOD _copyFromModel_McStopProcess
  VAR_IN_OUT
    {attribute 'OPC.UA.DA' := '0'}
    model : M_McStopProcess;
  END_VAR
                  THIS^.set := model.set;
SUPER^._copyFromModel_BaseMcProcess( model := model );

                
END_METHOD

METHOD _copyToModel_McStopProcess
  VAR_IN_OUT
    {attribute 'OPC.UA.DA' := '0'}
    model : M_McStopProcess;
  END_VAR
                  model.set := THIS^.set;
SUPER^._copyToModel_BaseMcProcess( model := model );

                
END_METHOD
END_FUNCTION_BLOCK

FUNCTION_BLOCK McMoveVelocityProcess EXTENDS BaseMcProcess
  VAR_INPUT
    {attribute 'OPC.UA.DA' := '1'}
    {attribute 'OPC.UA.DA.Access' := '3'}
    {attribute 'TcHmiSymbol.Show'}
    set : McMoveVelocityProcessArgs;  (* Arguments to be set, before writing do_request TRUE *)
  END_VAR
  VAR_OUTPUT
    {attribute 'OPC.UA.DA' := '0'}
    get : McMoveVelocityProcessArgs;  (* Arguments in use by the process, if do_request was accepted *)
  END_VAR

            IF do_request OR atomic.request THEN
    do_request_result := request( value := set.value );
    do_request := FALSE;
    atomic.request := FALSE;
END_IF;
SUPER^();

          

{attribute 'TcRpcEnable' := '1'}
METHOD start
  VAR_INPUT
    value : LREAL;  (* New velocity *)
  END_VAR
                  THIS^.get.value := value;
IF THIS^.atomic.request THEN
    THIS^.stat.handle := THIS^.atomic.handle;
ELSE
    THIS^.stat.handle := 0;
END_IF;
THIS^.stat.busy := BusyStatus.busy;
THIS^.stat.health := HealthStatus.good;

                
END_METHOD

{attribute 'TcRpcEnable' := '1'}
METHOD request : RequestResults
  VAR_INPUT
    value : LREAL;  (* New velocity *)
  END_VAR
                  IF THIS^.stat.enabled = EnabledStatus.enabled THEN
    request := RequestResults.ACCEPTED;
    THIS^.start( value := value );
ELSE
    request := RequestResults.REJECTED;
    IF THIS^.atomic.request THEN
        THIS^.lastRejectedHandle := THIS^.atomic.handle;
    END_IF;
END_IF;

                
END_METHOD

METHOD _copyFromModel_McMoveVelocityProcess
  VAR_IN_OUT
    {attribute 'OPC.UA.DA' := '0'}
    model : M_McMoveVelocityProcess;
  END_VAR
                  THIS^.set := model.set;
SUPER^._copyFromModel_BaseMcProcess( model := model );

                
END_METHOD

METHOD _copyToModel_McMoveVelocityProcess
  VAR_IN_OUT
    {attribute 'OPC.UA.DA' := '0'}
    model : M_McMoveVelocityProcess;
  END_VAR
                  model.set := THIS^.set;
SUPER^._copyToModel_BaseMcProcess( model := model );

                
END_METHOD
END_FUNCTION_BLOCK

FUNCTION_BLOCK SetEnabledProcess EXTENDS BaseProcess
  VAR_INPUT
    {attribute 'OPC.UA.DA' := '1'}
    {attribute 'OPC.UA.DA.Access' := '3'}
    {attribute 'TcHmiSymbol.Show'}
    set : SetEnabledProcessArgs;  (* Arguments to be set, before writing do_request TRUE *)
  END_VAR
  VAR_OUTPUT
    {attribute 'OPC.UA.DA' := '0'}
    get : SetEnabledProcessArgs;  (* Arguments in use by the process, if do_request was accepted *)
  END_VAR

            IF do_request OR atomic.request THEN
    do_request_result := request( enabled := set.enabled );
    do_request := FALSE;
    atomic.request := FALSE;
END_IF;
SUPER^();

          

{attribute 'TcRpcEnable' := '1'}
METHOD start
  VAR_INPUT
    enabled : BOOL;  (* True to enable, false to disable *)
  END_VAR
                  THIS^.get.enabled := enabled;
IF THIS^.atomic.request THEN
    THIS^.stat.handle := THIS^.atomic.handle;
ELSE
    THIS^.stat.handle := 0;
END_IF;
THIS^.stat.busy := BusyStatus.busy;
THIS^.stat.health := HealthStatus.good;

                
END_METHOD

{attribute 'TcRpcEnable' := '1'}
METHOD request : RequestResults
  VAR_INPUT
    enabled : BOOL;  (* True to enable, false to disable *)
  END_VAR
                  IF THIS^.stat.enabled = EnabledStatus.enabled THEN
    request := RequestResults.ACCEPTED;
    THIS^.start( enabled := enabled );
ELSE
    request := RequestResults.REJECTED;
    IF THIS^.atomic.request THEN
        THIS^.lastRejectedHandle := THIS^.atomic.handle;
    END_IF;
END_IF;

                
END_METHOD

METHOD _copyFromModel_SetEnabledProcess
  VAR_IN_OUT
    {attribute 'OPC.UA.DA' := '0'}
    model : M_SetEnabledProcess;
  END_VAR
                  THIS^.set := model.set;
SUPER^._copyFromModel_BaseProcess( model := model );

                
END_METHOD

METHOD _copyToModel_SetEnabledProcess
  VAR_IN_OUT
    {attribute 'OPC.UA.DA' := '0'}
    model : M_SetEnabledProcess;
  END_VAR
                  model.set := THIS^.set;
SUPER^._copyToModel_BaseProcess( model := model );

                
END_METHOD
END_FUNCTION_BLOCK

FUNCTION_BLOCK McWriteParameter EXTENDS BaseMcProcess
  VAR_INPUT
    {attribute 'OPC.UA.DA' := '1'}
    {attribute 'OPC.UA.DA.Access' := '3'}
    {attribute 'TcHmiSymbol.Show'}
    set : McWriteParameterArgs;  (* Arguments to be set, before writing do_request TRUE *)
  END_VAR
  VAR_OUTPUT
    {attribute 'OPC.UA.DA' := '0'}
    get : McWriteParameterArgs;  (* Arguments in use by the process, if do_request was accepted *)
  END_VAR

            IF do_request OR atomic.request THEN
    do_request_result := request(
    parameterNumber := set.parameterNumber,
    value := set.value);
    do_request := FALSE;
    atomic.request := FALSE;
END_IF;
SUPER^();

          

{attribute 'TcRpcEnable' := '1'}
METHOD start
  VAR_INPUT
    parameterNumber : INT;  (* Number of the parameter *)
    value : LREAL;  (* Value to write *)
  END_VAR
                  THIS^.get.parameterNumber := parameterNumber;
THIS^.get.value := value;
IF THIS^.atomic.request THEN
    THIS^.stat.handle := THIS^.atomic.handle;
ELSE
    THIS^.stat.handle := 0;
END_IF;
THIS^.stat.busy := BusyStatus.busy;
THIS^.stat.health := HealthStatus.good;

                
END_METHOD

{attribute 'TcRpcEnable' := '1'}
METHOD request : RequestResults
  VAR_INPUT
    parameterNumber : INT;  (* Number of the parameter *)
    value : LREAL;  (* Value to write *)
  END_VAR
                  IF THIS^.stat.enabled = EnabledStatus.enabled THEN
    request := RequestResults.ACCEPTED;
    THIS^.start(
        parameterNumber := parameterNumber,
        value := value);
ELSE
    request := RequestResults.REJECTED;
    IF THIS^.atomic.request THEN
        THIS^.lastRejectedHandle := THIS^.atomic.handle;
    END_IF;
END_IF;

                
END_METHOD

METHOD _copyFromModel_McWriteParameter
  VAR_IN_OUT
    {attribute 'OPC.UA.DA' := '0'}
    model : M_McWriteParameter;
  END_VAR
                  THIS^.set := model.set;
SUPER^._copyFromModel_BaseMcProcess( model := model );

                
END_METHOD

METHOD _copyToModel_McWriteParameter
  VAR_IN_OUT
    {attribute 'OPC.UA.DA' := '0'}
    model : M_McWriteParameter;
  END_VAR
                  model.set := THIS^.set;
SUPER^._copyToModel_BaseMcProcess( model := model );

                
END_METHOD
END_FUNCTION_BLOCK

FUNCTION_BLOCK McReadParameter EXTENDS BaseMcProcess
  VAR_INPUT
    {attribute 'OPC.UA.DA' := '1'}
    value : LREAL;  (* Value that was read *)
    {attribute 'OPC.UA.DA' := '1'}
    {attribute 'OPC.UA.DA.Access' := '3'}
    {attribute 'TcHmiSymbol.Show'}
    set : McReadParameterArgs;  (* Arguments to be set, before writing do_request TRUE *)
  END_VAR
  VAR_OUTPUT
    {attribute 'OPC.UA.DA' := '0'}
    get : McReadParameterArgs;  (* Arguments in use by the process, if do_request was accepted *)
  END_VAR

            IF do_request OR atomic.request THEN
    do_request_result := request( parameterNumber := set.parameterNumber );
    do_request := FALSE;
    atomic.request := FALSE;
END_IF;
SUPER^();

          

{attribute 'TcRpcEnable' := '1'}
METHOD start
  VAR_INPUT
    parameterNumber : INT;  (* Number of the parameter *)
  END_VAR
                  THIS^.get.parameterNumber := parameterNumber;
IF THIS^.atomic.request THEN
    THIS^.stat.handle := THIS^.atomic.handle;
ELSE
    THIS^.stat.handle := 0;
END_IF;
THIS^.stat.busy := BusyStatus.busy;
THIS^.stat.health := HealthStatus.good;

                
END_METHOD

{attribute 'TcRpcEnable' := '1'}
METHOD request : RequestResults
  VAR_INPUT
    parameterNumber : INT;  (* Number of the parameter *)
  END_VAR
                  IF THIS^.stat.enabled = EnabledStatus.enabled THEN
    request := RequestResults.ACCEPTED;
    THIS^.start( parameterNumber := parameterNumber );
ELSE
    request := RequestResults.REJECTED;
    IF THIS^.atomic.request THEN
        THIS^.lastRejectedHandle := THIS^.atomic.handle;
    END_IF;
END_IF;

                
END_METHOD

METHOD _copyFromModel_McReadParameter
  VAR_IN_OUT
    {attribute 'OPC.UA.DA' := '0'}
    model : M_McReadParameter;
  END_VAR
                  THIS^.set := model.set;
SUPER^._copyFromModel_BaseMcProcess( model := model );

                
END_METHOD

METHOD _copyToModel_McReadParameter
  VAR_IN_OUT
    {attribute 'OPC.UA.DA' := '0'}
    model : M_McReadParameter;
  END_VAR
                  model.value := THIS^.value;
model.set := THIS^.set;
SUPER^._copyToModel_BaseMcProcess( model := model );

                
END_METHOD
END_FUNCTION_BLOCK

FUNCTION_BLOCK McWriteBoolParameter EXTENDS BaseMcProcess
  VAR_INPUT
    {attribute 'OPC.UA.DA' := '1'}
    {attribute 'OPC.UA.DA.Access' := '3'}
    {attribute 'TcHmiSymbol.Show'}
    set : McWriteBoolParameterArgs;  (* Arguments to be set, before writing do_request TRUE *)
  END_VAR
  VAR_OUTPUT
    {attribute 'OPC.UA.DA' := '0'}
    get : McWriteBoolParameterArgs;  (* Arguments in use by the process, if do_request was accepted *)
  END_VAR

            IF do_request OR atomic.request THEN
    do_request_result := request(
    parameterNumber := set.parameterNumber,
    value := set.value);
    do_request := FALSE;
    atomic.request := FALSE;
END_IF;
SUPER^();

          

{attribute 'TcRpcEnable' := '1'}
METHOD start
  VAR_INPUT
    parameterNumber : INT;  (* Number of the parameter *)
    value : BOOL;  (* Value to write *)
  END_VAR
                  THIS^.get.parameterNumber := parameterNumber;
THIS^.get.value := value;
IF THIS^.atomic.request THEN
    THIS^.stat.handle := THIS^.atomic.handle;
ELSE
    THIS^.stat.handle := 0;
END_IF;
THIS^.stat.busy := BusyStatus.busy;
THIS^.stat.health := HealthStatus.good;

                
END_METHOD

{attribute 'TcRpcEnable' := '1'}
METHOD request : RequestResults
  VAR_INPUT
    parameterNumber : INT;  (* Number of the parameter *)
    value : BOOL;  (* Value to write *)
  END_VAR
                  IF THIS^.stat.enabled = EnabledStatus.enabled THEN
    request := RequestResults.ACCEPTED;
    THIS^.start(
        parameterNumber := parameterNumber,
        value := value);
ELSE
    request := RequestResults.REJECTED;
    IF THIS^.atomic.request THEN
        THIS^.lastRejectedHandle := THIS^.atomic.handle;
    END_IF;
END_IF;

                
END_METHOD

METHOD _copyFromModel_McWriteBoolParameter
  VAR_IN_OUT
    {attribute 'OPC.UA.DA' := '0'}
    model : M_McWriteBoolParameter;
  END_VAR
                  THIS^.set := model.set;
SUPER^._copyFromModel_BaseMcProcess( model := model );

                
END_METHOD

METHOD _copyToModel_McWriteBoolParameter
  VAR_IN_OUT
    {attribute 'OPC.UA.DA' := '0'}
    model : M_McWriteBoolParameter;
  END_VAR
                  model.set := THIS^.set;
SUPER^._copyToModel_BaseMcProcess( model := model );

                
END_METHOD
END_FUNCTION_BLOCK

FUNCTION_BLOCK McReadBoolParameter EXTENDS BaseMcProcess
  VAR_INPUT
    {attribute 'OPC.UA.DA' := '1'}
    value : BOOL;  (* Value that was read *)
    {attribute 'OPC.UA.DA' := '1'}
    {attribute 'OPC.UA.DA.Access' := '3'}
    {attribute 'TcHmiSymbol.Show'}
    set : McReadBoolParameterArgs;  (* Arguments to be set, before writing do_request TRUE *)
  END_VAR
  VAR_OUTPUT
    {attribute 'OPC.UA.DA' := '0'}
    get : McReadBoolParameterArgs;  (* Arguments in use by the process, if do_request was accepted *)
  END_VAR

            IF do_request OR atomic.request THEN
    do_request_result := request( parameterNumber := set.parameterNumber );
    do_request := FALSE;
    atomic.request := FALSE;
END_IF;
SUPER^();

          

{attribute 'TcRpcEnable' := '1'}
METHOD start
  VAR_INPUT
    parameterNumber : INT;  (* Number of the parameter *)
  END_VAR
                  THIS^.get.parameterNumber := parameterNumber;
IF THIS^.atomic.request THEN
    THIS^.stat.handle := THIS^.atomic.handle;
ELSE
    THIS^.stat.handle := 0;
END_IF;
THIS^.stat.busy := BusyStatus.busy;
THIS^.stat.health := HealthStatus.good;

                
END_METHOD

{attribute 'TcRpcEnable' := '1'}
METHOD request : RequestResults
  VAR_INPUT
    parameterNumber : INT;  (* Number of the parameter *)
  END_VAR
                  IF THIS^.stat.enabled = EnabledStatus.enabled THEN
    request := RequestResults.ACCEPTED;
    THIS^.start( parameterNumber := parameterNumber );
ELSE
    request := RequestResults.REJECTED;
    IF THIS^.atomic.request THEN
        THIS^.lastRejectedHandle := THIS^.atomic.handle;
    END_IF;
END_IF;

                
END_METHOD

METHOD _copyFromModel_McReadBoolParameter
  VAR_IN_OUT
    {attribute 'OPC.UA.DA' := '0'}
    model : M_McReadBoolParameter;
  END_VAR
                  THIS^.set := model.set;
SUPER^._copyFromModel_BaseMcProcess( model := model );

                
END_METHOD

METHOD _copyToModel_McReadBoolParameter
  VAR_IN_OUT
    {attribute 'OPC.UA.DA' := '0'}
    model : M_McReadBoolParameter;
  END_VAR
                  model.value := THIS^.value;
model.set := THIS^.set;
SUPER^._copyToModel_BaseMcProcess( model := model );

                
END_METHOD
END_FUNCTION_BLOCK

FUNCTION_BLOCK McProbe EXTENDS BaseMcProcess
  VAR_INPUT
    {attribute 'OPC.UA.DA' := '1'}
    recordedPosition : LREAL;  (* Value that was probed *)
    {attribute 'OPC.UA.DA' := '1'}
    {attribute 'OPC.UA.DA.Access' := '3'}
    {attribute 'TcHmiSymbol.Show'}
    set : McProbeArgs;  (* Arguments to be set, before writing do_request TRUE *)
  END_VAR
  VAR_OUTPUT
    {attribute 'OPC.UA.DA' := '0'}
    get : McProbeArgs;  (* Arguments in use by the process, if do_request was accepted *)
  END_VAR

            IF do_request OR atomic.request THEN
    do_request_result := request(
    risingEdge := set.risingEdge,
    timeout := set.timeout);
    do_request := FALSE;
    atomic.request := FALSE;
END_IF;
SUPER^();

          

{attribute 'TcRpcEnable' := '1'}
METHOD start
  VAR_INPUT
    risingEdge : BOOL;  (* True to probe the rising edge, false to probe the falling edge *)
    timeout : LREAL;  (* Timeout, in seconds. After this timeout, probing is aborted. timeout <= 0 means endless probing. *)
  END_VAR
                  THIS^.get.risingEdge := risingEdge;
THIS^.get.timeout := timeout;
IF THIS^.atomic.request THEN
    THIS^.stat.handle := THIS^.atomic.handle;
ELSE
    THIS^.stat.handle := 0;
END_IF;
THIS^.stat.busy := BusyStatus.busy;
THIS^.stat.health := HealthStatus.good;

                
END_METHOD

{attribute 'TcRpcEnable' := '1'}
METHOD request : RequestResults
  VAR_INPUT
    risingEdge : BOOL;  (* True to probe the rising edge, false to probe the falling edge *)
    timeout : LREAL;  (* Timeout, in seconds. After this timeout, probing is aborted. timeout <= 0 means endless probing. *)
  END_VAR
                  IF THIS^.stat.enabled = EnabledStatus.enabled THEN
    request := RequestResults.ACCEPTED;
    THIS^.start(
        risingEdge := risingEdge,
        timeout := timeout);
ELSE
    request := RequestResults.REJECTED;
    IF THIS^.atomic.request THEN
        THIS^.lastRejectedHandle := THIS^.atomic.handle;
    END_IF;
END_IF;

                
END_METHOD

METHOD _copyFromModel_McProbe
  VAR_IN_OUT
    {attribute 'OPC.UA.DA' := '0'}
    model : M_McProbe;
  END_VAR
                  THIS^.set := model.set;
SUPER^._copyFromModel_BaseMcProcess( model := model );

                
END_METHOD

METHOD _copyToModel_McProbe
  VAR_IN_OUT
    {attribute 'OPC.UA.DA' := '0'}
    model : M_McProbe;
  END_VAR
                  model.recordedPosition := THIS^.recordedPosition;
model.set := THIS^.set;
SUPER^._copyToModel_BaseMcProcess( model := model );

                
END_METHOD
END_FUNCTION_BLOCK

FUNCTION_BLOCK ChangeOperatingStateProcess EXTENDS BaseProcess
  VAR_INPUT
    {attribute 'OPC.UA.DA' := '1'}
    {attribute 'OPC.UA.DA.Access' := '3'}
    {attribute 'TcHmiSymbol.Show'}
    set : ChangeOperatingStateProcessArgs;  (* Arguments to be set, before writing do_request TRUE *)
  END_VAR
  VAR_OUTPUT
    {attribute 'OPC.UA.DA' := '0'}
    get : ChangeOperatingStateProcessArgs;  (* Arguments in use by the process, if do_request was accepted *)
  END_VAR

            IF do_request OR atomic.request THEN
    do_request_result := request( state := set.state );
    do_request := FALSE;
    atomic.request := FALSE;
END_IF;
SUPER^();

          

{attribute 'TcRpcEnable' := '1'}
METHOD start
  VAR_INPUT
    state : OperatingStates;  (* New operating state (e.g. AUTO, MANUAL) *)
  END_VAR
                  THIS^.get.state := state;
IF THIS^.atomic.request THEN
    THIS^.stat.handle := THIS^.atomic.handle;
ELSE
    THIS^.stat.handle := 0;
END_IF;
THIS^.stat.busy := BusyStatus.busy;
THIS^.stat.health := HealthStatus.good;

                
END_METHOD

{attribute 'TcRpcEnable' := '1'}
METHOD request : RequestResults
  VAR_INPUT
    state : OperatingStates;  (* New operating state (e.g. AUTO, MANUAL) *)
  END_VAR
                  IF THIS^.stat.enabled = EnabledStatus.enabled THEN
    request := RequestResults.ACCEPTED;
    THIS^.start( state := state );
ELSE
    request := RequestResults.REJECTED;
    IF THIS^.atomic.request THEN
        THIS^.lastRejectedHandle := THIS^.atomic.handle;
    END_IF;
END_IF;

                
END_METHOD

METHOD _copyFromModel_ChangeOperatingStateProcess
  VAR_IN_OUT
    {attribute 'OPC.UA.DA' := '0'}
    model : M_ChangeOperatingStateProcess;
  END_VAR
                  THIS^.set := model.set;
SUPER^._copyFromModel_BaseProcess( model := model );

                
END_METHOD

METHOD _copyToModel_ChangeOperatingStateProcess
  VAR_IN_OUT
    {attribute 'OPC.UA.DA' := '0'}
    model : M_ChangeOperatingStateProcess;
  END_VAR
                  model.set := THIS^.set;
SUPER^._copyToModel_BaseProcess( model := model );

                
END_METHOD
END_FUNCTION_BLOCK

FUNCTION_BLOCK ChangeOperatorStateProcess EXTENDS BaseProcess
  VAR_INPUT
    {attribute 'OPC.UA.DA' := '1'}
    {attribute 'OPC.UA.DA.Access' := '3'}
    {attribute 'TcHmiSymbol.Show'}
    set : ChangeOperatorStateProcessArgs;  (* Arguments to be set, before writing do_request TRUE *)
  END_VAR
  VAR_OUTPUT
    {attribute 'OPC.UA.DA' := '0'}
    get : ChangeOperatorStateProcessArgs;  (* Arguments in use by the process, if do_request was accepted *)
  END_VAR

            IF do_request OR atomic.request THEN
    do_request_result := request(
    state := set.state,
    password := set.password);
    do_request := FALSE;
    atomic.request := FALSE;
END_IF;
SUPER^();

          

{attribute 'TcRpcEnable' := '1'}
METHOD start
  VAR_INPUT
    state : OperatorStates;  (* New operator state (e.g. OBSERVER, TECH, ...) *)
    password : STRING(12);  (* Password (only sometimes required, e.g. to go from OBSERVER to TECH) *)
  END_VAR
                  THIS^.get.state := state;
THIS^.get.password := password;
IF THIS^.atomic.request THEN
    THIS^.stat.handle := THIS^.atomic.handle;
ELSE
    THIS^.stat.handle := 0;
END_IF;
THIS^.stat.busy := BusyStatus.busy;
THIS^.stat.health := HealthStatus.good;

                
END_METHOD

{attribute 'TcRpcEnable' := '1'}
METHOD request : RequestResults
  VAR_INPUT
    state : OperatorStates;  (* New operator state (e.g. OBSERVER, TECH, ...) *)
    password : STRING(12);  (* Password (only sometimes required, e.g. to go from OBSERVER to TECH) *)
  END_VAR
                  IF THIS^.stat.enabled = EnabledStatus.enabled THEN
    request := RequestResults.ACCEPTED;
    THIS^.start(
        state := state,
        password := password);
ELSE
    request := RequestResults.REJECTED;
    IF THIS^.atomic.request THEN
        THIS^.lastRejectedHandle := THIS^.atomic.handle;
    END_IF;
END_IF;

                
END_METHOD

METHOD _copyFromModel_ChangeOperatorStateProcess
  VAR_IN_OUT
    {attribute 'OPC.UA.DA' := '0'}
    model : M_ChangeOperatorStateProcess;
  END_VAR
                  THIS^.set := model.set;
SUPER^._copyFromModel_BaseProcess( model := model );

                
END_METHOD

METHOD _copyToModel_ChangeOperatorStateProcess
  VAR_IN_OUT
    {attribute 'OPC.UA.DA' := '0'}
    model : M_ChangeOperatorStateProcess;
  END_VAR
                  model.set := THIS^.set;
SUPER^._copyToModel_BaseProcess( model := model );

                
END_METHOD
END_FUNCTION_BLOCK

FUNCTION_BLOCK ChangeOperatingModeStateProcess EXTENDS BaseProcess
  VAR_INPUT
    {attribute 'OPC.UA.DA' := '1'}
    {attribute 'OPC.UA.DA.Access' := '3'}
    {attribute 'TcHmiSymbol.Show'}
    set : ChangeOperatingModeStateProcessArgs;  (* Arguments to be set, before writing do_request TRUE *)
  END_VAR
  VAR_OUTPUT
    {attribute 'OPC.UA.DA' := '0'}
    get : ChangeOperatingModeStateProcessArgs;  (* Arguments in use by the process, if do_request was accepted *)
  END_VAR

            IF do_request OR atomic.request THEN
    do_request_result := request( state := set.state );
    do_request := FALSE;
    atomic.request := FALSE;
END_IF;
SUPER^();

          

{attribute 'TcRpcEnable' := '1'}
METHOD start
  VAR_INPUT
    state : OperatingModeStates;  (* New operating state (e.g. LOCAL, REMOTE) *)
  END_VAR
                  THIS^.get.state := state;
IF THIS^.atomic.request THEN
    THIS^.stat.handle := THIS^.atomic.handle;
ELSE
    THIS^.stat.handle := 0;
END_IF;
THIS^.stat.busy := BusyStatus.busy;
THIS^.stat.health := HealthStatus.good;

                
END_METHOD

{attribute 'TcRpcEnable' := '1'}
METHOD request : RequestResults
  VAR_INPUT
    state : OperatingModeStates;  (* New operating state (e.g. LOCAL, REMOTE) *)
  END_VAR
                  IF THIS^.stat.enabled = EnabledStatus.enabled THEN
    request := RequestResults.ACCEPTED;
    THIS^.start( state := state );
ELSE
    request := RequestResults.REJECTED;
    IF THIS^.atomic.request THEN
        THIS^.lastRejectedHandle := THIS^.atomic.handle;
    END_IF;
END_IF;

                
END_METHOD

METHOD _copyFromModel_ChangeOperatingModeStateProcess
  VAR_IN_OUT
    {attribute 'OPC.UA.DA' := '0'}
    model : M_ChangeOperatingModeStateProcess;
  END_VAR
                  THIS^.set := model.set;
SUPER^._copyFromModel_BaseProcess( model := model );

                
END_METHOD

METHOD _copyToModel_ChangeOperatingModeStateProcess
  VAR_IN_OUT
    {attribute 'OPC.UA.DA' := '0'}
    model : M_ChangeOperatingModeStateProcess;
  END_VAR
                  model.set := THIS^.set;
SUPER^._copyToModel_BaseProcess( model := model );

                
END_METHOD
END_FUNCTION_BLOCK

FUNCTION_BLOCK ReadXmlProcess EXTENDS BaseXmlDataSrvProcess
  VAR_INPUT
    {attribute 'OPC.UA.DA' := '1'}
    {attribute 'OPC.UA.DA.Access' := '3'}
    {attribute 'TcHmiSymbol.Show'}
    set : ReadXmlProcessArgs;  (* Arguments to be set, before writing do_request TRUE *)
  END_VAR
  VAR_OUTPUT
    {attribute 'OPC.UA.DA' := '0'}
    get : ReadXmlProcessArgs;  (* Arguments in use by the process, if do_request was accepted *)
  END_VAR

            IF do_request OR atomic.request THEN
    do_request_result := request( filePath := set.filePath );
    do_request := FALSE;
    atomic.request := FALSE;
END_IF;
SUPER^();

          

{attribute 'TcRpcEnable' := '1'}
METHOD start
  VAR_INPUT
    filePath : STRING(30);  (* Full path of the filename to read *)
  END_VAR
                  THIS^.get.filePath := filePath;
IF THIS^.atomic.request THEN
    THIS^.stat.handle := THIS^.atomic.handle;
ELSE
    THIS^.stat.handle := 0;
END_IF;
THIS^.stat.busy := BusyStatus.busy;
THIS^.stat.health := HealthStatus.good;

                
END_METHOD

{attribute 'TcRpcEnable' := '1'}
METHOD request : RequestResults
  VAR_INPUT
    filePath : STRING(30);  (* Full path of the filename to read *)
  END_VAR
                  IF THIS^.stat.enabled = EnabledStatus.enabled THEN
    request := RequestResults.ACCEPTED;
    THIS^.start( filePath := filePath );
ELSE
    request := RequestResults.REJECTED;
    IF THIS^.atomic.request THEN
        THIS^.lastRejectedHandle := THIS^.atomic.handle;
    END_IF;
END_IF;

                
END_METHOD

METHOD _copyFromModel_ReadXmlProcess
  VAR_IN_OUT
    {attribute 'OPC.UA.DA' := '0'}
    model : M_ReadXmlProcess;
  END_VAR
                  THIS^.set := model.set;
SUPER^._copyFromModel_BaseXmlDataSrvProcess( model := model );

                
END_METHOD

METHOD _copyToModel_ReadXmlProcess
  VAR_IN_OUT
    {attribute 'OPC.UA.DA' := '0'}
    model : M_ReadXmlProcess;
  END_VAR
                  model.set := THIS^.set;
SUPER^._copyToModel_BaseXmlDataSrvProcess( model := model );

                
END_METHOD
END_FUNCTION_BLOCK

FUNCTION_BLOCK WriteXmlProcess EXTENDS BaseXmlDataSrvProcess
  VAR_INPUT
    {attribute 'OPC.UA.DA' := '1'}
    {attribute 'OPC.UA.DA.Access' := '3'}
    {attribute 'TcHmiSymbol.Show'}
    set : WriteXmlProcessArgs;  (* Arguments to be set, before writing do_request TRUE *)
  END_VAR
  VAR_OUTPUT
    {attribute 'OPC.UA.DA' := '0'}
    get : WriteXmlProcessArgs;  (* Arguments in use by the process, if do_request was accepted *)
  END_VAR

            IF do_request OR atomic.request THEN
    do_request_result := request( filePath := set.filePath );
    do_request := FALSE;
    atomic.request := FALSE;
END_IF;
SUPER^();

          

{attribute 'TcRpcEnable' := '1'}
METHOD start
  VAR_INPUT
    filePath : STRING(30);  (* Full path of the filename to write *)
  END_VAR
                  THIS^.get.filePath := filePath;
IF THIS^.atomic.request THEN
    THIS^.stat.handle := THIS^.atomic.handle;
ELSE
    THIS^.stat.handle := 0;
END_IF;
THIS^.stat.busy := BusyStatus.busy;
THIS^.stat.health := HealthStatus.good;

                
END_METHOD

{attribute 'TcRpcEnable' := '1'}
METHOD request : RequestResults
  VAR_INPUT
    filePath : STRING(30);  (* Full path of the filename to write *)
  END_VAR
                  IF THIS^.stat.enabled = EnabledStatus.enabled THEN
    request := RequestResults.ACCEPTED;
    THIS^.start( filePath := filePath );
ELSE
    request := RequestResults.REJECTED;
    IF THIS^.atomic.request THEN
        THIS^.lastRejectedHandle := THIS^.atomic.handle;
    END_IF;
END_IF;

                
END_METHOD

METHOD _copyFromModel_WriteXmlProcess
  VAR_IN_OUT
    {attribute 'OPC.UA.DA' := '0'}
    model : M_WriteXmlProcess;
  END_VAR
                  THIS^.set := model.set;
SUPER^._copyFromModel_BaseXmlDataSrvProcess( model := model );

                
END_METHOD

METHOD _copyToModel_WriteXmlProcess
  VAR_IN_OUT
    {attribute 'OPC.UA.DA' := '0'}
    model : M_WriteXmlProcess;
  END_VAR
                  model.set := THIS^.set;
SUPER^._copyToModel_BaseXmlDataSrvProcess( model := model );

                
END_METHOD
END_FUNCTION_BLOCK

FUNCTION_BLOCK ActivateProcess EXTENDS BaseProcess

            IF do_request OR atomic.request THEN
    do_request_result := request();
    do_request := FALSE;
    atomic.request := FALSE;
END_IF;
SUPER^();

          

{attribute 'TcRpcEnable' := '1'}
METHOD start
                  IF THIS^.atomic.request THEN
    THIS^.stat.handle := THIS^.atomic.handle;
ELSE
    THIS^.stat.handle := 0;
END_IF;
THIS^.stat.busy := BusyStatus.busy;
THIS^.stat.health := HealthStatus.good;

                
END_METHOD

{attribute 'TcRpcEnable' := '1'}
METHOD request : RequestResults
                  IF THIS^.stat.enabled = EnabledStatus.enabled THEN
    request := RequestResults.ACCEPTED;
    THIS^.start();
ELSE
    request := RequestResults.REJECTED;
    IF THIS^.atomic.request THEN
        THIS^.lastRejectedHandle := THIS^.atomic.handle;
    END_IF;
END_IF;

                
END_METHOD

METHOD _copyFromModel_ActivateProcess
  VAR_IN_OUT
    {attribute 'OPC.UA.DA' := '0'}
    model : M_ActivateProcess;
  END_VAR
                  SUPER^._copyFromModel_BaseProcess( model := model );

                
END_METHOD

METHOD _copyToModel_ActivateProcess
  VAR_IN_OUT
    {attribute 'OPC.UA.DA' := '0'}
    model : M_ActivateProcess;
  END_VAR
                  SUPER^._copyToModel_BaseProcess( model := model );

                
END_METHOD
END_FUNCTION_BLOCK

FUNCTION_BLOCK ModbusRTUBusReadCoilProcess EXTENDS BaseProcess
  VAR_INPUT
    {attribute 'OPC.UA.DA' := '1'}
    value : BOOL;  (* Value of the coil *)
    {attribute 'OPC.UA.DA' := '1'}
    errorId : INT;  (* Error Id. Modbus error code *)
    {attribute 'OPC.UA.DA' := '1'}
    {attribute 'OPC.UA.DA.Access' := '3'}
    {attribute 'TcHmiSymbol.Show'}
    set : ModbusRTUBusReadCoilProcessArgs;  (* Arguments to be set, before writing do_request TRUE *)
  END_VAR
  VAR_OUTPUT
    {attribute 'OPC.UA.DA' := '0'}
    get : ModbusRTUBusReadCoilProcessArgs;  (* Arguments in use by the process, if do_request was accepted *)
  END_VAR

            IF do_request OR atomic.request THEN
    do_request_result := request(
    unitID := set.unitID,
    address := set.address);
    do_request := FALSE;
    atomic.request := FALSE;
END_IF;
SUPER^();

          

{attribute 'TcRpcEnable' := '1'}
METHOD start
  VAR_INPUT
    unitID : USINT;  (* Modbus station address (1..247) *)
    address : UINT;  (* Modbus data address *)
  END_VAR
                  THIS^.get.unitID := unitID;
THIS^.get.address := address;
IF THIS^.atomic.request THEN
    THIS^.stat.handle := THIS^.atomic.handle;
ELSE
    THIS^.stat.handle := 0;
END_IF;
THIS^.stat.busy := BusyStatus.busy;
THIS^.stat.health := HealthStatus.good;

                
END_METHOD

{attribute 'TcRpcEnable' := '1'}
METHOD request : RequestResults
  VAR_INPUT
    unitID : USINT;  (* Modbus station address (1..247) *)
    address : UINT;  (* Modbus data address *)
  END_VAR
                  IF THIS^.stat.enabled = EnabledStatus.enabled THEN
    request := RequestResults.ACCEPTED;
    THIS^.start(
        unitID := unitID,
        address := address);
ELSE
    request := RequestResults.REJECTED;
    IF THIS^.atomic.request THEN
        THIS^.lastRejectedHandle := THIS^.atomic.handle;
    END_IF;
END_IF;

                
END_METHOD

METHOD _copyFromModel_ModbusRTUBusReadCoilProcess
  VAR_IN_OUT
    {attribute 'OPC.UA.DA' := '0'}
    model : M_ModbusRTUBusReadCoilProcess;
  END_VAR
                  THIS^.set := model.set;
SUPER^._copyFromModel_BaseProcess( model := model );

                
END_METHOD

METHOD _copyToModel_ModbusRTUBusReadCoilProcess
  VAR_IN_OUT
    {attribute 'OPC.UA.DA' := '0'}
    model : M_ModbusRTUBusReadCoilProcess;
  END_VAR
                  model.value := THIS^.value;
model.errorId := THIS^.errorId;
model.set := THIS^.set;
SUPER^._copyToModel_BaseProcess( model := model );

                
END_METHOD
END_FUNCTION_BLOCK

FUNCTION_BLOCK ModbusRTUBusWriteCoilProcess EXTENDS BaseProcess
  VAR_INPUT
    {attribute 'OPC.UA.DA' := '1'}
    errorId : INT;  (* Error Id. Modbus error code *)
    {attribute 'OPC.UA.DA' := '1'}
    {attribute 'OPC.UA.DA.Access' := '3'}
    {attribute 'TcHmiSymbol.Show'}
    set : ModbusRTUBusWriteCoilProcessArgs;  (* Arguments to be set, before writing do_request TRUE *)
  END_VAR
  VAR_OUTPUT
    {attribute 'OPC.UA.DA' := '0'}
    get : ModbusRTUBusWriteCoilProcessArgs;  (* Arguments in use by the process, if do_request was accepted *)
  END_VAR

            IF do_request OR atomic.request THEN
    do_request_result := request(
    unitID := set.unitID,
    address := set.address,
    value := set.value);
    do_request := FALSE;
    atomic.request := FALSE;
END_IF;
SUPER^();

          

{attribute 'TcRpcEnable' := '1'}
METHOD start
  VAR_INPUT
    unitID : USINT;  (* Modbus station address (1..247) *)
    address : UINT;  (* Modbus data address *)
    value : BOOL;  (* Value to write on the coil *)
  END_VAR
                  THIS^.get.unitID := unitID;
THIS^.get.address := address;
THIS^.get.value := value;
IF THIS^.atomic.request THEN
    THIS^.stat.handle := THIS^.atomic.handle;
ELSE
    THIS^.stat.handle := 0;
END_IF;
THIS^.stat.busy := BusyStatus.busy;
THIS^.stat.health := HealthStatus.good;

                
END_METHOD

{attribute 'TcRpcEnable' := '1'}
METHOD request : RequestResults
  VAR_INPUT
    unitID : USINT;  (* Modbus station address (1..247) *)
    address : UINT;  (* Modbus data address *)
    value : BOOL;  (* Value to write on the coil *)
  END_VAR
                  IF THIS^.stat.enabled = EnabledStatus.enabled THEN
    request := RequestResults.ACCEPTED;
    THIS^.start(
        unitID := unitID,
        address := address,
        value := value);
ELSE
    request := RequestResults.REJECTED;
    IF THIS^.atomic.request THEN
        THIS^.lastRejectedHandle := THIS^.atomic.handle;
    END_IF;
END_IF;

                
END_METHOD

METHOD _copyFromModel_ModbusRTUBusWriteCoilProcess
  VAR_IN_OUT
    {attribute 'OPC.UA.DA' := '0'}
    model : M_ModbusRTUBusWriteCoilProcess;
  END_VAR
                  THIS^.set := model.set;
SUPER^._copyFromModel_BaseProcess( model := model );

                
END_METHOD

METHOD _copyToModel_ModbusRTUBusWriteCoilProcess
  VAR_IN_OUT
    {attribute 'OPC.UA.DA' := '0'}
    model : M_ModbusRTUBusWriteCoilProcess;
  END_VAR
                  model.errorId := THIS^.errorId;
model.set := THIS^.set;
SUPER^._copyToModel_BaseProcess( model := model );

                
END_METHOD
END_FUNCTION_BLOCK

FUNCTION_BLOCK ModbusRTUBusReadRegisterProcess EXTENDS BaseProcess
  VAR_INPUT
    {attribute 'OPC.UA.DA' := '1'}
    value : INT;  (* Value of the register *)
    {attribute 'OPC.UA.DA' := '1'}
    errorId : INT;  (* Error Id. Modbus error code *)
    {attribute 'OPC.UA.DA' := '1'}
    {attribute 'OPC.UA.DA.Access' := '3'}
    {attribute 'TcHmiSymbol.Show'}
    set : ModbusRTUBusReadRegisterProcessArgs;  (* Arguments to be set, before writing do_request TRUE *)
  END_VAR
  VAR_OUTPUT
    {attribute 'OPC.UA.DA' := '0'}
    get : ModbusRTUBusReadRegisterProcessArgs;  (* Arguments in use by the process, if do_request was accepted *)
  END_VAR

            IF do_request OR atomic.request THEN
    do_request_result := request(
    unitID := set.unitID,
    address := set.address);
    do_request := FALSE;
    atomic.request := FALSE;
END_IF;
SUPER^();

          

{attribute 'TcRpcEnable' := '1'}
METHOD start
  VAR_INPUT
    unitID : USINT;  (* Modbus station address (1..247) *)
    address : UINT;  (* Modbus data address *)
  END_VAR
                  THIS^.get.unitID := unitID;
THIS^.get.address := address;
IF THIS^.atomic.request THEN
    THIS^.stat.handle := THIS^.atomic.handle;
ELSE
    THIS^.stat.handle := 0;
END_IF;
THIS^.stat.busy := BusyStatus.busy;
THIS^.stat.health := HealthStatus.good;

                
END_METHOD

{attribute 'TcRpcEnable' := '1'}
METHOD request : RequestResults
  VAR_INPUT
    unitID : USINT;  (* Modbus station address (1..247) *)
    address : UINT;  (* Modbus data address *)
  END_VAR
                  IF THIS^.stat.enabled = EnabledStatus.enabled THEN
    request := RequestResults.ACCEPTED;
    THIS^.start(
        unitID := unitID,
        address := address);
ELSE
    request := RequestResults.REJECTED;
    IF THIS^.atomic.request THEN
        THIS^.lastRejectedHandle := THIS^.atomic.handle;
    END_IF;
END_IF;

                
END_METHOD

METHOD _copyFromModel_ModbusRTUBusReadRegisterProcess
  VAR_IN_OUT
    {attribute 'OPC.UA.DA' := '0'}
    model : M_ModbusRTUBusReadRegisterProcess;
  END_VAR
                  THIS^.set := model.set;
SUPER^._copyFromModel_BaseProcess( model := model );

                
END_METHOD

METHOD _copyToModel_ModbusRTUBusReadRegisterProcess
  VAR_IN_OUT
    {attribute 'OPC.UA.DA' := '0'}
    model : M_ModbusRTUBusReadRegisterProcess;
  END_VAR
                  model.value := THIS^.value;
model.errorId := THIS^.errorId;
model.set := THIS^.set;
SUPER^._copyToModel_BaseProcess( model := model );

                
END_METHOD
END_FUNCTION_BLOCK

FUNCTION_BLOCK ModbusRTUBusWriteRegisterProcess EXTENDS BaseProcess
  VAR_INPUT
    {attribute 'OPC.UA.DA' := '1'}
    errorId : INT;  (* Error Id. Modbus error code *)
    {attribute 'OPC.UA.DA' := '1'}
    {attribute 'OPC.UA.DA.Access' := '3'}
    {attribute 'TcHmiSymbol.Show'}
    set : ModbusRTUBusWriteRegisterProcessArgs;  (* Arguments to be set, before writing do_request TRUE *)
  END_VAR
  VAR_OUTPUT
    {attribute 'OPC.UA.DA' := '0'}
    get : ModbusRTUBusWriteRegisterProcessArgs;  (* Arguments in use by the process, if do_request was accepted *)
  END_VAR

            IF do_request OR atomic.request THEN
    do_request_result := request(
    unitID := set.unitID,
    address := set.address,
    value := set.value);
    do_request := FALSE;
    atomic.request := FALSE;
END_IF;
SUPER^();

          

{attribute 'TcRpcEnable' := '1'}
METHOD start
  VAR_INPUT
    unitID : USINT;  (* Modbus station address (1..247) *)
    address : UINT;  (* Modbus data address *)
    value : INT;  (* Value to write on the register *)
  END_VAR
                  THIS^.get.unitID := unitID;
THIS^.get.address := address;
THIS^.get.value := value;
IF THIS^.atomic.request THEN
    THIS^.stat.handle := THIS^.atomic.handle;
ELSE
    THIS^.stat.handle := 0;
END_IF;
THIS^.stat.busy := BusyStatus.busy;
THIS^.stat.health := HealthStatus.good;

                
END_METHOD

{attribute 'TcRpcEnable' := '1'}
METHOD request : RequestResults
  VAR_INPUT
    unitID : USINT;  (* Modbus station address (1..247) *)
    address : UINT;  (* Modbus data address *)
    value : INT;  (* Value to write on the register *)
  END_VAR
                  IF THIS^.stat.enabled = EnabledStatus.enabled THEN
    request := RequestResults.ACCEPTED;
    THIS^.start(
        unitID := unitID,
        address := address,
        value := value);
ELSE
    request := RequestResults.REJECTED;
    IF THIS^.atomic.request THEN
        THIS^.lastRejectedHandle := THIS^.atomic.handle;
    END_IF;
END_IF;

                
END_METHOD

METHOD _copyFromModel_ModbusRTUBusWriteRegisterProcess
  VAR_IN_OUT
    {attribute 'OPC.UA.DA' := '0'}
    model : M_ModbusRTUBusWriteRegisterProcess;
  END_VAR
                  THIS^.set := model.set;
SUPER^._copyFromModel_BaseProcess( model := model );

                
END_METHOD

METHOD _copyToModel_ModbusRTUBusWriteRegisterProcess
  VAR_IN_OUT
    {attribute 'OPC.UA.DA' := '0'}
    model : M_ModbusRTUBusWriteRegisterProcess;
  END_VAR
                  model.errorId := THIS^.errorId;
model.set := THIS^.set;
SUPER^._copyToModel_BaseProcess( model := model );

                
END_METHOD
END_FUNCTION_BLOCK

FUNCTION_BLOCK ModbusRTUBusDiagnosticsProcess EXTENDS BaseProcess
  VAR_INPUT
    {attribute 'OPC.UA.DA' := '1'}
    value : INT;  (* Value of the register *)
    {attribute 'OPC.UA.DA' := '1'}
    errorId : INT;  (* Error Id. Modbus error code *)
    {attribute 'OPC.UA.DA' := '1'}
    {attribute 'OPC.UA.DA.Access' := '3'}
    {attribute 'TcHmiSymbol.Show'}
    set : ModbusRTUBusDiagnosticsProcessArgs;  (* Arguments to be set, before writing do_request TRUE *)
  END_VAR
  VAR_OUTPUT
    {attribute 'OPC.UA.DA' := '0'}
    get : ModbusRTUBusDiagnosticsProcessArgs;  (* Arguments in use by the process, if do_request was accepted *)
  END_VAR

            IF do_request OR atomic.request THEN
    do_request_result := request(
    unitID := set.unitID,
    subFunction := set.subFunction,
    subData := set.subData);
    do_request := FALSE;
    atomic.request := FALSE;
END_IF;
SUPER^();

          

{attribute 'TcRpcEnable' := '1'}
METHOD start
  VAR_INPUT
    unitID : USINT;  (* Modbus station address (1..247) *)
    subFunction : UINT;  (* Modbus subFunction code *)
    subData : INT;  (* Modbus data for subFunction *)
  END_VAR
                  THIS^.get.unitID := unitID;
THIS^.get.subFunction := subFunction;
THIS^.get.subData := subData;
IF THIS^.atomic.request THEN
    THIS^.stat.handle := THIS^.atomic.handle;
ELSE
    THIS^.stat.handle := 0;
END_IF;
THIS^.stat.busy := BusyStatus.busy;
THIS^.stat.health := HealthStatus.good;

                
END_METHOD

{attribute 'TcRpcEnable' := '1'}
METHOD request : RequestResults
  VAR_INPUT
    unitID : USINT;  (* Modbus station address (1..247) *)
    subFunction : UINT;  (* Modbus subFunction code *)
    subData : INT;  (* Modbus data for subFunction *)
  END_VAR
                  IF THIS^.stat.enabled = EnabledStatus.enabled THEN
    request := RequestResults.ACCEPTED;
    THIS^.start(
        unitID := unitID,
        subFunction := subFunction,
        subData := subData);
ELSE
    request := RequestResults.REJECTED;
    IF THIS^.atomic.request THEN
        THIS^.lastRejectedHandle := THIS^.atomic.handle;
    END_IF;
END_IF;

                
END_METHOD

METHOD _copyFromModel_ModbusRTUBusDiagnosticsProcess
  VAR_IN_OUT
    {attribute 'OPC.UA.DA' := '0'}
    model : M_ModbusRTUBusDiagnosticsProcess;
  END_VAR
                  THIS^.set := model.set;
SUPER^._copyFromModel_BaseProcess( model := model );

                
END_METHOD

METHOD _copyToModel_ModbusRTUBusDiagnosticsProcess
  VAR_IN_OUT
    {attribute 'OPC.UA.DA' := '0'}
    model : M_ModbusRTUBusDiagnosticsProcess;
  END_VAR
                  model.value := THIS^.value;
model.errorId := THIS^.errorId;
model.set := THIS^.set;
SUPER^._copyToModel_BaseProcess( model := model );

                
END_METHOD
END_FUNCTION_BLOCK

FUNCTION_BLOCK PointAlphaDeltaProcess EXTENDS BaseProcess
  VAR_INPUT
    {attribute 'OPC.UA.DA' := '1'}
    {attribute 'OPC.UA.DA.Access' := '3'}
    {attribute 'TcHmiSymbol.Show'}
    set : PointAlphaDeltaProcessArgs;  (* Arguments to be set, before writing do_request TRUE *)
  END_VAR
  VAR_OUTPUT
    {attribute 'OPC.UA.DA' := '0'}
    get : PointAlphaDeltaProcessArgs;  (* Arguments in use by the process, if do_request was accepted *)
  END_VAR

            IF do_request OR atomic.request THEN
    do_request_result := request(
    alpha := set.alpha,
    delta := set.delta);
    do_request := FALSE;
    atomic.request := FALSE;
END_IF;
SUPER^();

          

{attribute 'TcRpcEnable' := '1'}
METHOD start
  VAR_INPUT
    alpha : LREAL;  (* Right ascention, in hours *)
    delta : LREAL;  (* Declination, in degrees *)
  END_VAR
                  THIS^.get.alpha := alpha;
THIS^.get.delta := delta;
IF THIS^.atomic.request THEN
    THIS^.stat.handle := THIS^.atomic.handle;
ELSE
    THIS^.stat.handle := 0;
END_IF;
THIS^.stat.busy := BusyStatus.busy;
THIS^.stat.health := HealthStatus.good;

                
END_METHOD

{attribute 'TcRpcEnable' := '1'}
METHOD request : RequestResults
  VAR_INPUT
    alpha : LREAL;  (* Right ascention, in hours *)
    delta : LREAL;  (* Declination, in degrees *)
  END_VAR
                  IF THIS^.stat.enabled = EnabledStatus.enabled THEN
    request := RequestResults.ACCEPTED;
    THIS^.start(
        alpha := alpha,
        delta := delta);
ELSE
    request := RequestResults.REJECTED;
    IF THIS^.atomic.request THEN
        THIS^.lastRejectedHandle := THIS^.atomic.handle;
    END_IF;
END_IF;

                
END_METHOD

METHOD _copyFromModel_PointAlphaDeltaProcess
  VAR_IN_OUT
    {attribute 'OPC.UA.DA' := '0'}
    model : M_PointAlphaDeltaProcess;
  END_VAR
                  THIS^.set := model.set;
SUPER^._copyFromModel_BaseProcess( model := model );

                
END_METHOD

METHOD _copyToModel_PointAlphaDeltaProcess
  VAR_IN_OUT
    {attribute 'OPC.UA.DA' := '0'}
    model : M_PointAlphaDeltaProcess;
  END_VAR
                  model.set := THIS^.set;
SUPER^._copyToModel_BaseProcess( model := model );

                
END_METHOD
END_FUNCTION_BLOCK

FUNCTION_BLOCK GigECameraSetParamProcess EXTENDS BaseProcess
  VAR_INPUT
    {attribute 'OPC.UA.DA' := '1'}
    {attribute 'OPC.UA.DA.Access' := '3'}
    {attribute 'TcHmiSymbol.Show'}
    set : GigECameraSetParamProcessArgs;  (* Arguments to be set, before writing do_request TRUE *)
  END_VAR
  VAR_OUTPUT
    {attribute 'OPC.UA.DA' := '0'}
    get : GigECameraSetParamProcessArgs;  (* Arguments in use by the process, if do_request was accepted *)
  END_VAR

            IF do_request OR atomic.request THEN
    do_request_result := request(
    param := set.param,
    nValue := set.nValue,
    fvalue := set.fvalue,
    refresh := set.refresh);
    do_request := FALSE;
    atomic.request := FALSE;
END_IF;
SUPER^();

          

{attribute 'TcRpcEnable' := '1'}
METHOD start
  VAR_INPUT
    param : GigECameraParams;  (* UInt32 Parameter *)
    nValue : UDINT;  (* Integer Value *)
    fvalue : LREAL;  (* Double Value *)
    refresh : BOOL := TRUE;  (* Refresh the parameter set after the write (slower!) *)
  END_VAR
                  THIS^.get.param := param;
THIS^.get.nValue := nValue;
THIS^.get.fvalue := fvalue;
THIS^.get.refresh := refresh;
IF THIS^.atomic.request THEN
    THIS^.stat.handle := THIS^.atomic.handle;
ELSE
    THIS^.stat.handle := 0;
END_IF;
THIS^.stat.busy := BusyStatus.busy;
THIS^.stat.health := HealthStatus.good;

                
END_METHOD

{attribute 'TcRpcEnable' := '1'}
METHOD request : RequestResults
  VAR_INPUT
    param : GigECameraParams;  (* UInt32 Parameter *)
    nValue : UDINT;  (* Integer Value *)
    fvalue : LREAL;  (* Double Value *)
    refresh : BOOL := TRUE;  (* Refresh the parameter set after the write (slower!) *)
  END_VAR
                  IF THIS^.stat.enabled = EnabledStatus.enabled THEN
    request := RequestResults.ACCEPTED;
    THIS^.start(
        param := param,
        nValue := nValue,
        fvalue := fvalue,
        refresh := refresh);
ELSE
    request := RequestResults.REJECTED;
    IF THIS^.atomic.request THEN
        THIS^.lastRejectedHandle := THIS^.atomic.handle;
    END_IF;
END_IF;

                
END_METHOD

METHOD _copyFromModel_GigECameraSetParamProcess
  VAR_IN_OUT
    {attribute 'OPC.UA.DA' := '0'}
    model : M_GigECameraSetParamProcess;
  END_VAR
                  THIS^.set := model.set;
SUPER^._copyFromModel_BaseProcess( model := model );

                
END_METHOD

METHOD _copyToModel_GigECameraSetParamProcess
  VAR_IN_OUT
    {attribute 'OPC.UA.DA' := '0'}
    model : M_GigECameraSetParamProcess;
  END_VAR
                  model.set := THIS^.set;
SUPER^._copyToModel_BaseProcess( model := model );

                
END_METHOD
END_FUNCTION_BLOCK

FUNCTION_BLOCK GigECameraSetParam2Process EXTENDS BaseProcess
  VAR_INPUT
    {attribute 'OPC.UA.DA' := '1'}
    {attribute 'OPC.UA.DA.Access' := '3'}
    {attribute 'TcHmiSymbol.Show'}
    set : GigECameraSetParam2ProcessArgs;  (* Arguments to be set, before writing do_request TRUE *)
  END_VAR
  VAR_OUTPUT
    {attribute 'OPC.UA.DA' := '0'}
    get : GigECameraSetParam2ProcessArgs;  (* Arguments in use by the process, if do_request was accepted *)
  END_VAR

            IF do_request OR atomic.request THEN
    do_request_result := request(
    param1 := set.param1,
    nValue1 := set.nValue1,
    fvalue1 := set.fvalue1,
    param2 := set.param2,
    nValue2 := set.nValue2,
    fvalue2 := set.fvalue2,
    refresh := set.refresh);
    do_request := FALSE;
    atomic.request := FALSE;
END_IF;
SUPER^();

          

{attribute 'TcRpcEnable' := '1'}
METHOD start
  VAR_INPUT
    param1 : GigECameraParams;  (* UInt32 Parameter 1 *)
    nValue1 : UDINT;  (* Integer Value of Parameter 1 *)
    fvalue1 : LREAL;  (* Double Value of Parameter 1 *)
    param2 : GigECameraParams;  (* UInt32 Parameter 2 *)
    nValue2 : UDINT;  (* Integer Value of Parameter 2 *)
    fvalue2 : LREAL;  (* Double Value of Parameter 2 *)
    refresh : BOOL := TRUE;  (* Refresh the parameter set after the write (slower!) *)
  END_VAR
                  THIS^.get.param1 := param1;
THIS^.get.nValue1 := nValue1;
THIS^.get.fvalue1 := fvalue1;
THIS^.get.param2 := param2;
THIS^.get.nValue2 := nValue2;
THIS^.get.fvalue2 := fvalue2;
THIS^.get.refresh := refresh;
IF THIS^.atomic.request THEN
    THIS^.stat.handle := THIS^.atomic.handle;
ELSE
    THIS^.stat.handle := 0;
END_IF;
THIS^.stat.busy := BusyStatus.busy;
THIS^.stat.health := HealthStatus.good;

                
END_METHOD

{attribute 'TcRpcEnable' := '1'}
METHOD request : RequestResults
  VAR_INPUT
    param1 : GigECameraParams;  (* UInt32 Parameter 1 *)
    nValue1 : UDINT;  (* Integer Value of Parameter 1 *)
    fvalue1 : LREAL;  (* Double Value of Parameter 1 *)
    param2 : GigECameraParams;  (* UInt32 Parameter 2 *)
    nValue2 : UDINT;  (* Integer Value of Parameter 2 *)
    fvalue2 : LREAL;  (* Double Value of Parameter 2 *)
    refresh : BOOL := TRUE;  (* Refresh the parameter set after the write (slower!) *)
  END_VAR
                  IF THIS^.stat.enabled = EnabledStatus.enabled THEN
    request := RequestResults.ACCEPTED;
    THIS^.start(
        param1 := param1,
        nValue1 := nValue1,
        fvalue1 := fvalue1,
        param2 := param2,
        nValue2 := nValue2,
        fvalue2 := fvalue2,
        refresh := refresh);
ELSE
    request := RequestResults.REJECTED;
    IF THIS^.atomic.request THEN
        THIS^.lastRejectedHandle := THIS^.atomic.handle;
    END_IF;
END_IF;

                
END_METHOD

METHOD _copyFromModel_GigECameraSetParam2Process
  VAR_IN_OUT
    {attribute 'OPC.UA.DA' := '0'}
    model : M_GigECameraSetParam2Process;
  END_VAR
                  THIS^.set := model.set;
SUPER^._copyFromModel_BaseProcess( model := model );

                
END_METHOD

METHOD _copyToModel_GigECameraSetParam2Process
  VAR_IN_OUT
    {attribute 'OPC.UA.DA' := '0'}
    model : M_GigECameraSetParam2Process;
  END_VAR
                  model.set := THIS^.set;
SUPER^._copyToModel_BaseProcess( model := model );

                
END_METHOD
END_FUNCTION_BLOCK

FUNCTION_BLOCK GigECameraPulseTrigger EXTENDS BaseProcess
  VAR_INPUT
    {attribute 'OPC.UA.DA' := '1'}
    {attribute 'OPC.UA.DA.Access' := '3'}
    {attribute 'TcHmiSymbol.Show'}
    set : GigECameraPulseTriggerArgs;  (* Arguments to be set, before writing do_request TRUE *)
  END_VAR
  VAR_OUTPUT
    {attribute 'OPC.UA.DA' := '0'}
    get : GigECameraPulseTriggerArgs;  (* Arguments in use by the process, if do_request was accepted *)
  END_VAR

            IF do_request OR atomic.request THEN
    do_request_result := request( duration := set.duration );
    do_request := FALSE;
    atomic.request := FALSE;
END_IF;
SUPER^();

          

{attribute 'TcRpcEnable' := '1'}
METHOD start
  VAR_INPUT
    duration : LREAL;  (* Duration in seconds of the pulse *)
  END_VAR
                  THIS^.get.duration := duration;
IF THIS^.atomic.request THEN
    THIS^.stat.handle := THIS^.atomic.handle;
ELSE
    THIS^.stat.handle := 0;
END_IF;
THIS^.stat.busy := BusyStatus.busy;
THIS^.stat.health := HealthStatus.good;

                
END_METHOD

{attribute 'TcRpcEnable' := '1'}
METHOD request : RequestResults
  VAR_INPUT
    duration : LREAL;  (* Duration in seconds of the pulse *)
  END_VAR
                  IF THIS^.stat.enabled = EnabledStatus.enabled THEN
    request := RequestResults.ACCEPTED;
    THIS^.start( duration := duration );
ELSE
    request := RequestResults.REJECTED;
    IF THIS^.atomic.request THEN
        THIS^.lastRejectedHandle := THIS^.atomic.handle;
    END_IF;
END_IF;

                
END_METHOD

METHOD _copyFromModel_GigECameraPulseTrigger
  VAR_IN_OUT
    {attribute 'OPC.UA.DA' := '0'}
    model : M_GigECameraPulseTrigger;
  END_VAR
                  THIS^.set := model.set;
SUPER^._copyFromModel_BaseProcess( model := model );

                
END_METHOD

METHOD _copyToModel_GigECameraPulseTrigger
  VAR_IN_OUT
    {attribute 'OPC.UA.DA' := '0'}
    model : M_GigECameraPulseTrigger;
  END_VAR
                  model.set := THIS^.set;
SUPER^._copyToModel_BaseProcess( model := model );

                
END_METHOD
END_FUNCTION_BLOCK

FUNCTION_BLOCK GigECameraSetSourceProcess EXTENDS BaseProcess
  VAR_INPUT
    {attribute 'OPC.UA.DA' := '1'}
    {attribute 'OPC.UA.DA.Access' := '3'}
    {attribute 'TcHmiSymbol.Show'}
    set : GigECameraSetSourceProcessArgs;  (* Arguments to be set, before writing do_request TRUE *)
  END_VAR
  VAR_OUTPUT
    {attribute 'OPC.UA.DA' := '0'}
    get : GigECameraSetSourceProcessArgs;  (* Arguments in use by the process, if do_request was accepted *)
  END_VAR

            IF do_request OR atomic.request THEN
    do_request_result := request( source := set.source );
    do_request := FALSE;
    atomic.request := FALSE;
END_IF;
SUPER^();

          

{attribute 'TcRpcEnable' := '1'}
METHOD start
  VAR_INPUT
    source : GigECameraSources;  (* Camera source to set *)
  END_VAR
                  THIS^.get.source := source;
IF THIS^.atomic.request THEN
    THIS^.stat.handle := THIS^.atomic.handle;
ELSE
    THIS^.stat.handle := 0;
END_IF;
THIS^.stat.busy := BusyStatus.busy;
THIS^.stat.health := HealthStatus.good;

                
END_METHOD

{attribute 'TcRpcEnable' := '1'}
METHOD request : RequestResults
  VAR_INPUT
    source : GigECameraSources;  (* Camera source to set *)
  END_VAR
                  IF THIS^.stat.enabled = EnabledStatus.enabled THEN
    request := RequestResults.ACCEPTED;
    THIS^.start( source := source );
ELSE
    request := RequestResults.REJECTED;
    IF THIS^.atomic.request THEN
        THIS^.lastRejectedHandle := THIS^.atomic.handle;
    END_IF;
END_IF;

                
END_METHOD

METHOD _copyFromModel_GigECameraSetSourceProcess
  VAR_IN_OUT
    {attribute 'OPC.UA.DA' := '0'}
    model : M_GigECameraSetSourceProcess;
  END_VAR
                  THIS^.set := model.set;
SUPER^._copyFromModel_BaseProcess( model := model );

                
END_METHOD

METHOD _copyToModel_GigECameraSetSourceProcess
  VAR_IN_OUT
    {attribute 'OPC.UA.DA' := '0'}
    model : M_GigECameraSetSourceProcess;
  END_VAR
                  model.set := THIS^.set;
SUPER^._copyToModel_BaseProcess( model := model );

                
END_METHOD
END_FUNCTION_BLOCK

FUNCTION_BLOCK GigECameraSetupProcess EXTENDS BaseProcess
  VAR_INPUT
    {attribute 'OPC.UA.DA' := '1'}
    {attribute 'OPC.UA.DA.Access' := '3'}
    {attribute 'TcHmiSymbol.Show'}
    set : GigECameraSetupProcessArgs;  (* Arguments to be set, before writing do_request TRUE *)
  END_VAR
  VAR_OUTPUT
    {attribute 'OPC.UA.DA' := '0'}
    get : GigECameraSetupProcessArgs;  (* Arguments in use by the process, if do_request was accepted *)
  END_VAR

            IF do_request OR atomic.request THEN
    do_request_result := request(
    doExposureTime := set.doExposureTime,
    exposureTime := set.exposureTime,
    doFrameRate := set.doFrameRate,
    frameRate := set.frameRate,
    doWindowXY := set.doWindowXY,
    windowX := set.windowX,
    windowY := set.windowY,
    doWindowWH := set.doWindowWH,
    windowWidth := set.windowWidth,
    windowHeight := set.windowHeight,
    doBinning := set.doBinning,
    binningX := set.binningX,
    binningY := set.binningY,
    doAnalogGain := set.doAnalogGain,
    analogGain := set.analogGain,
    doDigitalGain := set.doDigitalGain,
    digitalGain := set.digitalGain,
    blackLevel := set.blackLevel,
    blackLevelAuto := set.blackLevelAuto,
    doBlackLevel := set.doBlackLevel,
    continuous := set.continuous,
    doContinuous := set.doContinuous);
    do_request := FALSE;
    atomic.request := FALSE;
END_IF;
SUPER^();

          

{attribute 'TcRpcEnable' := '1'}
METHOD start
  VAR_INPUT
    doExposureTime : BOOL := TRUE;  (* If TRUE, set the exposure time *)
    exposureTime : LREAL;  (* Exposure time in seconds *)
    doFrameRate : BOOL;  (* If TRUE, set the acquisition frame rate *)
    frameRate : LREAL;  (* Acquisition frame rate in Hz *)
    doWindowXY : BOOL;  (* If TRUE, set the window XY position *)
    windowX : UDINT;  (* Window X position in pixels *)
    windowY : UDINT;  (* Window Y position in pixels *)
    doWindowWH : BOOL;  (* If TRUE, set the window width and height *)
    windowWidth : UDINT;  (* Window width in pixels *)
    windowHeight : UDINT;  (* Window height in pixels *)
    doBinning : BOOL;  (* If TRUE, set the binning *)
    binningX : UDINT;  (* Binning X factor *)
    binningY : UDINT;  (* Binning Y factor *)
    doAnalogGain : BOOL;  (* If TRUE, set the analog gain *)
    analogGain : LREAL;  (* Analog gain *)
    doDigitalGain : BOOL;  (* If TRUE, set the digital gain *)
    digitalGain : LREAL;  (* Digital gain *)
    blackLevel : LREAL;  (* Black level (0 .. 511 for 12-bit images) *)
    blackLevelAuto : BOOL;  (* If TRUE, black level is set automatically. If FALSE, black level is set manually *)
    doBlackLevel : BOOL;  (* If TRUE, set the black level and black level auto *)
    continuous : BOOL;  (* If TRUE, set the continuous acquisition mode, trigger mode, etc. to continuous imaging *)
    doContinuous : BOOL;  (* If TRUE, set the continuous acquisition mode, trigger mode, etc. *)
  END_VAR
                  THIS^.get.doExposureTime := doExposureTime;
THIS^.get.exposureTime := exposureTime;
THIS^.get.doFrameRate := doFrameRate;
THIS^.get.frameRate := frameRate;
THIS^.get.doWindowXY := doWindowXY;
THIS^.get.windowX := windowX;
THIS^.get.windowY := windowY;
THIS^.get.doWindowWH := doWindowWH;
THIS^.get.windowWidth := windowWidth;
THIS^.get.windowHeight := windowHeight;
THIS^.get.doBinning := doBinning;
THIS^.get.binningX := binningX;
THIS^.get.binningY := binningY;
THIS^.get.doAnalogGain := doAnalogGain;
THIS^.get.analogGain := analogGain;
THIS^.get.doDigitalGain := doDigitalGain;
THIS^.get.digitalGain := digitalGain;
THIS^.get.blackLevel := blackLevel;
THIS^.get.blackLevelAuto := blackLevelAuto;
THIS^.get.doBlackLevel := doBlackLevel;
THIS^.get.continuous := continuous;
THIS^.get.doContinuous := doContinuous;
IF THIS^.atomic.request THEN
    THIS^.stat.handle := THIS^.atomic.handle;
ELSE
    THIS^.stat.handle := 0;
END_IF;
THIS^.stat.busy := BusyStatus.busy;
THIS^.stat.health := HealthStatus.good;

                
END_METHOD

{attribute 'TcRpcEnable' := '1'}
METHOD request : RequestResults
  VAR_INPUT
    doExposureTime : BOOL := TRUE;  (* If TRUE, set the exposure time *)
    exposureTime : LREAL;  (* Exposure time in seconds *)
    doFrameRate : BOOL;  (* If TRUE, set the acquisition frame rate *)
    frameRate : LREAL;  (* Acquisition frame rate in Hz *)
    doWindowXY : BOOL;  (* If TRUE, set the window XY position *)
    windowX : UDINT;  (* Window X position in pixels *)
    windowY : UDINT;  (* Window Y position in pixels *)
    doWindowWH : BOOL;  (* If TRUE, set the window width and height *)
    windowWidth : UDINT;  (* Window width in pixels *)
    windowHeight : UDINT;  (* Window height in pixels *)
    doBinning : BOOL;  (* If TRUE, set the binning *)
    binningX : UDINT;  (* Binning X factor *)
    binningY : UDINT;  (* Binning Y factor *)
    doAnalogGain : BOOL;  (* If TRUE, set the analog gain *)
    analogGain : LREAL;  (* Analog gain *)
    doDigitalGain : BOOL;  (* If TRUE, set the digital gain *)
    digitalGain : LREAL;  (* Digital gain *)
    blackLevel : LREAL;  (* Black level (0 .. 511 for 12-bit images) *)
    blackLevelAuto : BOOL;  (* If TRUE, black level is set automatically. If FALSE, black level is set manually *)
    doBlackLevel : BOOL;  (* If TRUE, set the black level and black level auto *)
    continuous : BOOL;  (* If TRUE, set the continuous acquisition mode, trigger mode, etc. to continuous imaging *)
    doContinuous : BOOL;  (* If TRUE, set the continuous acquisition mode, trigger mode, etc. *)
  END_VAR
                  IF THIS^.stat.enabled = EnabledStatus.enabled THEN
    request := RequestResults.ACCEPTED;
    THIS^.start(
        doExposureTime := doExposureTime,
        exposureTime := exposureTime,
        doFrameRate := doFrameRate,
        frameRate := frameRate,
        doWindowXY := doWindowXY,
        windowX := windowX,
        windowY := windowY,
        doWindowWH := doWindowWH,
        windowWidth := windowWidth,
        windowHeight := windowHeight,
        doBinning := doBinning,
        binningX := binningX,
        binningY := binningY,
        doAnalogGain := doAnalogGain,
        analogGain := analogGain,
        doDigitalGain := doDigitalGain,
        digitalGain := digitalGain,
        blackLevel := blackLevel,
        blackLevelAuto := blackLevelAuto,
        doBlackLevel := doBlackLevel,
        continuous := continuous,
        doContinuous := doContinuous);
ELSE
    request := RequestResults.REJECTED;
    IF THIS^.atomic.request THEN
        THIS^.lastRejectedHandle := THIS^.atomic.handle;
    END_IF;
END_IF;

                
END_METHOD

METHOD _copyFromModel_GigECameraSetupProcess
  VAR_IN_OUT
    {attribute 'OPC.UA.DA' := '0'}
    model : M_GigECameraSetupProcess;
  END_VAR
                  THIS^.set := model.set;
SUPER^._copyFromModel_BaseProcess( model := model );

                
END_METHOD

METHOD _copyToModel_GigECameraSetupProcess
  VAR_IN_OUT
    {attribute 'OPC.UA.DA' := '0'}
    model : M_GigECameraSetupProcess;
  END_VAR
                  model.set := THIS^.set;
SUPER^._copyToModel_BaseProcess( model := model );

                
END_METHOD
END_FUNCTION_BLOCK

FUNCTION_BLOCK GigECameraMultiTriggerProcess EXTENDS BaseProcess
  VAR_INPUT
    {attribute 'OPC.UA.DA' := '1'}
    {attribute 'OPC.UA.DA.Access' := '3'}
    {attribute 'TcHmiSymbol.Show'}
    set : GigECameraMultiTriggerProcessArgs;  (* Arguments to be set, before writing do_request TRUE *)
  END_VAR
  VAR_OUTPUT
    {attribute 'OPC.UA.DA' := '0'}
    get : GigECameraMultiTriggerProcessArgs;  (* Arguments in use by the process, if do_request was accepted *)
  END_VAR

            IF do_request OR atomic.request THEN
    do_request_result := request(
    count := set.count,
    algo := set.algo);
    do_request := FALSE;
    atomic.request := FALSE;
END_IF;
SUPER^();

          

{attribute 'TcRpcEnable' := '1'}
METHOD start
  VAR_INPUT
    count : UDINT;  (* Number of triggers to send *)
    algo : GigECameraMultiTriggerAlgorithms;  (* Algorithm to use for the multi-trigger *)
  END_VAR
                  THIS^.get.count := count;
THIS^.get.algo := algo;
IF THIS^.atomic.request THEN
    THIS^.stat.handle := THIS^.atomic.handle;
ELSE
    THIS^.stat.handle := 0;
END_IF;
THIS^.stat.busy := BusyStatus.busy;
THIS^.stat.health := HealthStatus.good;

                
END_METHOD

{attribute 'TcRpcEnable' := '1'}
METHOD request : RequestResults
  VAR_INPUT
    count : UDINT;  (* Number of triggers to send *)
    algo : GigECameraMultiTriggerAlgorithms;  (* Algorithm to use for the multi-trigger *)
  END_VAR
                  IF THIS^.stat.enabled = EnabledStatus.enabled THEN
    request := RequestResults.ACCEPTED;
    THIS^.start(
        count := count,
        algo := algo);
ELSE
    request := RequestResults.REJECTED;
    IF THIS^.atomic.request THEN
        THIS^.lastRejectedHandle := THIS^.atomic.handle;
    END_IF;
END_IF;

                
END_METHOD

METHOD _copyFromModel_GigECameraMultiTriggerProcess
  VAR_IN_OUT
    {attribute 'OPC.UA.DA' := '0'}
    model : M_GigECameraMultiTriggerProcess;
  END_VAR
                  THIS^.set := model.set;
SUPER^._copyFromModel_BaseProcess( model := model );

                
END_METHOD

METHOD _copyToModel_GigECameraMultiTriggerProcess
  VAR_IN_OUT
    {attribute 'OPC.UA.DA' := '0'}
    model : M_GigECameraMultiTriggerProcess;
  END_VAR
                  model.set := THIS^.set;
SUPER^._copyToModel_BaseProcess( model := model );

                
END_METHOD
END_FUNCTION_BLOCK

FUNCTION_BLOCK Arg1LrealProcess EXTENDS BaseProcess
  VAR_INPUT
    {attribute 'OPC.UA.DA' := '1'}
    {attribute 'OPC.UA.DA.Access' := '3'}
    {attribute 'TcHmiSymbol.Show'}
    set : Arg1LrealProcessArgs;  (* Arguments to be set, before writing do_request TRUE *)
  END_VAR
  VAR_OUTPUT
    {attribute 'OPC.UA.DA' := '0'}
    get : Arg1LrealProcessArgs;  (* Arguments in use by the process, if do_request was accepted *)
  END_VAR

            IF do_request OR atomic.request THEN
    do_request_result := request( setpoint := set.setpoint );
    do_request := FALSE;
    atomic.request := FALSE;
END_IF;
SUPER^();

          

{attribute 'TcRpcEnable' := '1'}
METHOD start
  VAR_INPUT
    setpoint : LREAL;  (* New setpoint value *)
  END_VAR
                  THIS^.get.setpoint := setpoint;
IF THIS^.atomic.request THEN
    THIS^.stat.handle := THIS^.atomic.handle;
ELSE
    THIS^.stat.handle := 0;
END_IF;
THIS^.stat.busy := BusyStatus.busy;
THIS^.stat.health := HealthStatus.good;

                
END_METHOD

{attribute 'TcRpcEnable' := '1'}
METHOD request : RequestResults
  VAR_INPUT
    setpoint : LREAL;  (* New setpoint value *)
  END_VAR
                  IF THIS^.stat.enabled = EnabledStatus.enabled THEN
    request := RequestResults.ACCEPTED;
    THIS^.start( setpoint := setpoint );
ELSE
    request := RequestResults.REJECTED;
    IF THIS^.atomic.request THEN
        THIS^.lastRejectedHandle := THIS^.atomic.handle;
    END_IF;
END_IF;

                
END_METHOD

METHOD _copyFromModel_Arg1LrealProcess
  VAR_IN_OUT
    {attribute 'OPC.UA.DA' := '0'}
    model : M_Arg1LrealProcess;
  END_VAR
                  THIS^.set := model.set;
SUPER^._copyFromModel_BaseProcess( model := model );

                
END_METHOD

METHOD _copyToModel_Arg1LrealProcess
  VAR_IN_OUT
    {attribute 'OPC.UA.DA' := '0'}
    model : M_Arg1LrealProcess;
  END_VAR
                  model.set := THIS^.set;
SUPER^._copyToModel_BaseProcess( model := model );

                
END_METHOD
END_FUNCTION_BLOCK

FUNCTION_BLOCK Ell114SendProcess EXTENDS BaseProcess
  VAR_INPUT
    {attribute 'OPC.UA.DA' := '1'}
    reply : STRING(20);  (* Raw reply by the stage *)
    {attribute 'OPC.UA.DA' := '1'}
    {attribute 'OPC.UA.DA.Access' := '3'}
    {attribute 'TcHmiSymbol.Show'}
    set : Ell114SendProcessArgs;  (* Arguments to be set, before writing do_request TRUE *)
  END_VAR
  VAR_OUTPUT
    {attribute 'OPC.UA.DA' := '0'}
    get : Ell114SendProcessArgs;  (* Arguments in use by the process, if do_request was accepted *)
  END_VAR

            IF do_request OR atomic.request THEN
    do_request_result := request(
    cmd := set.cmd,
    arg := set.arg);
    do_request := FALSE;
    atomic.request := FALSE;
END_IF;
SUPER^();

          

{attribute 'TcRpcEnable' := '1'}
METHOD start
  VAR_INPUT
    cmd : ELL14Command;  (* The command to be sent *)
    arg : STRING(10);  (* The payload of the command to be sent (excluding '0gs' or similar header, excluding $R$N suffix). Custom commands must include the header! *)
  END_VAR
                  THIS^.get.cmd := cmd;
THIS^.get.arg := arg;
IF THIS^.atomic.request THEN
    THIS^.stat.handle := THIS^.atomic.handle;
ELSE
    THIS^.stat.handle := 0;
END_IF;
THIS^.stat.busy := BusyStatus.busy;
THIS^.stat.health := HealthStatus.good;

                
END_METHOD

{attribute 'TcRpcEnable' := '1'}
METHOD request : RequestResults
  VAR_INPUT
    cmd : ELL14Command;  (* The command to be sent *)
    arg : STRING(10);  (* The payload of the command to be sent (excluding '0gs' or similar header, excluding $R$N suffix). Custom commands must include the header! *)
  END_VAR
                  IF THIS^.stat.enabled = EnabledStatus.enabled THEN
    request := RequestResults.ACCEPTED;
    THIS^.start(
        cmd := cmd,
        arg := arg);
ELSE
    request := RequestResults.REJECTED;
    IF THIS^.atomic.request THEN
        THIS^.lastRejectedHandle := THIS^.atomic.handle;
    END_IF;
END_IF;

                
END_METHOD

METHOD _copyFromModel_Ell114SendProcess
  VAR_IN_OUT
    {attribute 'OPC.UA.DA' := '0'}
    model : M_Ell114SendProcess;
  END_VAR
                  THIS^.set := model.set;
SUPER^._copyFromModel_BaseProcess( model := model );

                
END_METHOD

METHOD _copyToModel_Ell114SendProcess
  VAR_IN_OUT
    {attribute 'OPC.UA.DA' := '0'}
    model : M_Ell114SendProcess;
  END_VAR
                  model.reply := THIS^.reply;
model.set := THIS^.set;
SUPER^._copyToModel_BaseProcess( model := model );

                
END_METHOD
END_FUNCTION_BLOCK
